LIN {X 0,Y 398.886,Z 784.107,A -85,B 0,C 180,E1 -11229.847,E2 -11229.847} C_VEL
LIN {X 0,Y 402.44,Z 816.531,A -85,B 0,C 180,E1 -11230.643,E2 -11230.643} C_VEL
LIN {X 0,Y 403.181,Z 824.962,A -85,B 0,C 180,E1 -11230.833,E2 -11230.833} C_VEL
LIN {X 0,Y 402.235,Z 895.243,A -85,B 0,C 180,E1 -11232.105,E2 -11232.105} C_VEL
LIN {X 0,Y 401.617,Z 908.446,A -85,B 0,C 180,E1 -11232.537,E2 -11232.537} C_VEL
LIN {X 0,Y 400.757,Z 921.743,A -85,B 0,C 180,E1 -11233.189,E2 -11233.189} C_VEL
LIN {X 0,Y 399.896,Z 932.958,A -85,B 0,C 180,E1 -11233.939,E2 -11233.939} C_VEL
LIN {X 0,Y 398.89,Z 944.652,A -85,B 0,C 180,E1 -11234.945,E2 -11234.945} C_VEL
LIN {X 0,Y 398.165,Z 954.79,A -85,B 0,C 180,E1 -11236.038,E2 -11236.038} C_VEL
LIN {X 0,Y 397.612,Z 963.944,A -85,B 0,C 180,E1 -11237.243,E2 -11237.243} C_VEL
LIN {X 0,Y 396.995,Z 971.973,A -85,B 0,C 180,E1 -11238.52,E2 -11238.52} C_VEL
LIN {X 0,Y 396.564,Z 979.861,A -85,B 0,C 180,E1 -11240.057,E2 -11240.057} C_VEL
LIN {X 0,Y 396.358,Z 987.17,A -85,B 0,C 180,E1 -11241.852,E2 -11241.852} C_VEL
LIN {X 0,Y 396.334,Z 991.594,A -85,B 0,C 180,E1 -11243.229,E2 -11243.229} C_VEL
LIN {X 0,Y 396.382,Z 995.807,A -85,B 0,C 180,E1 -11244.921,E2 -11244.921} C_VEL
LIN {X 0,Y 396.495,Z 997.753,A -85,B 0,C 180,E1 -11245.941,E2 -11245.941} C_VEL
LIN {X 0,Y 396.453,Z 999.193,A -85,B 0,C 180,E1 -11246.958,E2 -11246.958} C_VEL
LIN {X 0,Y 396.473,Z 1000.227,A -85,B 0,C 180,E1 -11247.975,E2 -11247.975} C_VEL
LIN {X 0,Y 396.505,Z 1000.858,A -85,B 0,C 180,E1 -11248.991,E2 -11248.991} C_VEL
LIN {X 0,Y 396.533,Z 1001.082,A -85,B 0,C 180,E1 -11250.007,E2 -11250.007} C_VEL
LIN {X 0,Y 396.505,Z 1000.85,A -85,B 0,C 180,E1 -11251.022,E2 -11251.022} C_VEL
LIN {X 0,Y 396.475,Z 1000.211,A -85,B 0,C 180,E1 -11252.038,E2 -11252.038} C_VEL
LIN {X 0,Y 396.455,Z 999.171,A -85,B 0,C 180,E1 -11253.055,E2 -11253.055} C_VEL
LIN {X 0,Y 396.499,Z 997.722,A -85,B 0,C 180,E1 -11254.072,E2 -11254.072} C_VEL
LIN {X 0,Y 396.305,Z 994.645,A -85,B 0,C 180,E1 -11255.604,E2 -11255.604} C_VEL
LIN {X 0,Y 396.296,Z 990.519,A -85,B 0,C 180,E1 -11257.137,E2 -11257.137} C_VEL
LIN {X 0,Y 396.416,Z 984.19,A -85,B 0,C 180,E1 -11258.93,E2 -11258.93} C_VEL
LIN {X 0,Y 396.65,Z 977.307,A -85,B 0,C 180,E1 -11260.47,E2 -11260.47} C_VEL
LIN {X 0,Y 397.201,Z 968.823,A -85,B 0,C 180,E1 -11262.005,E2 -11262.005} C_VEL
LIN {X 0,Y 397.865,Z 960.153,A -85,B 0,C 180,E1 -11263.282,E2 -11263.282} C_VEL
LIN {X 0,Y 398.568,Z 950.667,A -85,B 0,C 180,E1 -11264.428,E2 -11264.428} C_VEL
LIN {X 0,Y 399.272,Z 940.375,A -85,B 0,C 180,E1 -11265.446,E2 -11265.446} C_VEL
LIN {X 0,Y 400.17,Z 929.216,A -85,B 0,C 180,E1 -11266.326,E2 -11266.326} C_VEL
LIN {X 0,Y 401.098,Z 916.885,A -85,B 0,C 180,E1 -11267.073,E2 -11267.073} C_VEL
LIN {X 0,Y 401.822,Z 903.894,A -85,B 0,C 180,E1 -11267.632,E2 -11267.632} C_VEL
LIN {X 0,Y 402.351,Z 890.094,A -85,B 0,C 180,E1 -11268.002,E2 -11268.002} C_VEL
LIN {X 0,Y 403.048,Z 822.221,A -85,B 0,C 180,E1 -11269.218,E2 -11269.218} C_VEL
LIN {X 0,Y 400.233,Z 790.769,A -85,B 0,C 180,E1 -11270.212,E2 -11270.212} C_VEL
LIN {X 0,Y 399.008,Z 781.49,A -85,B 0,C 180,E1 -11270.565,E2 -11270.565} C_VEL
LIN {X 0,Y 400.608,Z 758.553,A -85,B 0,C 180,E1 -11274.181,E2 -11274.181} C_VEL
LIN {X 0,Y 402.329,Z 735.168,A -85,B 0,C 180,E1 -11277.863,E2 -11277.863} C_VEL
LIN {X 0,Y 402.724,Z 728.077,A -85,B 0,C 180,E1 -11278.999,E2 -11278.999} C_VEL
LIN {X 0,Y 399.691,Z 713.868,A -85,B 0,C 180,E1 -11281.546,E2 -11281.546} C_VEL
LIN {X 0,Y 397.055,Z 703.027,A -85,B 0,C 180,E1 -11283.615,E2 -11283.615} C_VEL
LIN {X 0,Y 397.093,Z 703.019,A -85,B 0,C 180,E1 -11287.208,E2 -11287.208} C_VEL
LIN {X 0,Y 397.072,Z 703.022,A -85,B 0,C 180,E1 -11290.44,E2 -11290.44} C_VEL
LIN {X 0,Y 397.058,Z 703.025,A -85,B 0,C 180,E1 -11293.66,E2 -11293.66} C_VEL
LIN {X 0,Y 397.108,Z 703.017,A -85,B 0,C 180,E1 -11296.526,E2 -11296.526} C_VEL
LIN {X 0,Y 397.104,Z 703.018,A -85,B 0,C 180,E1 -11300.422,E2 -11300.422} C_VEL
LIN {X 0,Y 397.111,Z 703.018,A -85,B 0,C 180,E1 -11303.006,E2 -11303.006} C_VEL
LIN {X 0,Y 397.13,Z 703.014,A -85,B 0,C 180,E1 -11306.728,E2 -11306.728} C_VEL
LIN {X 0,Y 397.135,Z 703.016,A -85,B 0,C 180,E1 -11310.297,E2 -11310.297} C_VEL
LIN {X 0,Y 397.104,Z 703.023,A -85,B 0,C 180,E1 -11313.739,E2 -11313.739} C_VEL
LIN {X 0,Y 397.121,Z 703.02,A -85,B 0,C 180,E1 -11317.086,E2 -11317.086} C_VEL
LIN {X 0,Y 397.139,Z 703.111,A -85,B 0,C 180,E1 -11319.435,E2 -11319.435} C_VEL
LIN {X 0,Y 398.123,Z 705.838,A -85,B 0,C 180,E1 -11319.602,E2 -11319.602} C_VEL
LIN {X 0,Y 402.78,Z 715.108,A -85,B 0,C 180,E1 -11320.252,E2 -11320.252} C_VEL
LIN {X 0,Y 405.375,Z 721.504,A -85,B 0,C 180,E1 -11320.626,E2 -11320.626} C_VEL
LIN {X 0,Y 403.629,Z 784.545,A -85,B 0,C 180,E1 -11322.161,E2 -11322.161} C_VEL
LIN {X 0,Y 403.565,Z 799.417,A -85,B 0,C 180,E1 -11322.681,E2 -11322.681} C_VEL
LIN {X 0,Y 403.241,Z 810.911,A -85,B 0,C 180,E1 -11323.268,E2 -11323.268} C_VEL
LIN {X 0,Y 402.848,Z 820.383,A -85,B 0,C 180,E1 -11323.886,E2 -11323.886} C_VEL
LIN {X 0,Y 402.399,Z 829.533,A -85,B 0,C 180,E1 -11324.622,E2 -11324.622} C_VEL
LIN {X 0,Y 401.801,Z 837.999,A -85,B 0,C 180,E1 -11325.437,E2 -11325.437} C_VEL
LIN {X 0,Y 401.36,Z 845.689,A -85,B 0,C 180,E1 -11326.326,E2 -11326.326} C_VEL
LIN {X 0,Y 400.76,Z 853.176,A -85,B 0,C 180,E1 -11327.337,E2 -11327.337} C_VEL
LIN {X 0,Y 400.089,Z 860.892,A -85,B 0,C 180,E1 -11328.602,E2 -11328.602} C_VEL
LIN {X 0,Y 399.508,Z 867.261,A -85,B 0,C 180,E1 -11329.868,E2 -11329.868} C_VEL
LIN {X 0,Y 399.059,Z 871.627,A -85,B 0,C 180,E1 -11330.88,E2 -11330.88} C_VEL
LIN {X 0,Y 398.612,Z 876.825,A -85,B 0,C 180,E1 -11332.401,E2 -11332.401} C_VEL
LIN {X 0,Y 397.936,Z 880.867,A -85,B 0,C 180,E1 -11333.917,E2 -11333.917} C_VEL
LIN {X 0,Y 397.839,Z 882.927,A -85,B 0,C 180,E1 -11334.933,E2 -11334.933} C_VEL
LIN {X 0,Y 397.507,Z 885.635,A -85,B 0,C 180,E1 -11336.96,E2 -11336.96} C_VEL
LIN {X 0,Y 397.313,Z 886.407,A -85,B 0,C 180,E1 -11337.973,E2 -11337.973} C_VEL
LIN {X 0,Y 397.23,Z 886.702,A -85,B 0,C 180,E1 -11338.986,E2 -11338.986} C_VEL
LIN {X 0,Y 397.162,Z 886.546,A -85,B 0,C 180,E1 -11340,E2 -11340} C_VEL
LIN {X 0,Y 397.162,Z 885.976,A -85,B 0,C 180,E1 -11341.014,E2 -11341.014} C_VEL
LIN {X 0,Y 396.969,Z 883.539,A -85,B 0,C 180,E1 -11343.045,E2 -11343.045} C_VEL
LIN {X 0,Y 397.213,Z 880.535,A -85,B 0,C 180,E1 -11344.567,E2 -11344.567} C_VEL
LIN {X 0,Y 397.481,Z 878.001,A -85,B 0,C 180,E1 -11345.581,E2 -11345.581} C_VEL
LIN {X 0,Y 397.666,Z 873.185,A -85,B 0,C 180,E1 -11347.106,E2 -11347.106} C_VEL
LIN {X 0,Y 398.012,Z 866.134,A -85,B 0,C 180,E1 -11348.821,E2 -11348.821} C_VEL
LIN {X 0,Y 398.382,Z 859.325,A -85,B 0,C 180,E1 -11350.161,E2 -11350.161} C_VEL
LIN {X 0,Y 398.726,Z 853.236,A -85,B 0,C 180,E1 -11351.18,E2 -11351.18} C_VEL
LIN {X 0,Y 399.083,Z 845.109,A -85,B 0,C 180,E1 -11352.329,E2 -11352.329} C_VEL
LIN {X 0,Y 399.579,Z 836.504,A -85,B 0,C 180,E1 -11353.347,E2 -11353.347} C_VEL
LIN {X 0,Y 399.983,Z 827.526,A -85,B 0,C 180,E1 -11354.24,E2 -11354.24} C_VEL
LIN {X 0,Y 400.347,Z 817.268,A -85,B 0,C 180,E1 -11355.081,E2 -11355.081} C_VEL
LIN {X 0,Y 400.669,Z 807.831,A -85,B 0,C 180,E1 -11355.711,E2 -11355.711} C_VEL
LIN {X 0,Y 400.901,Z 796.867,A -85,B 0,C 180,E1 -11356.289,E2 -11356.289} C_VEL
LIN {X 0,Y 401.134,Z 786.297,A -85,B 0,C 180,E1 -11356.705,E2 -11356.705} C_VEL
LIN {X 0,Y 401.245,Z 773.112,A -85,B 0,C 180,E1 -11357.061,E2 -11357.061} C_VEL
LIN {X 0,Y 402.038,Z 717.884,A -85,B 0,C 180,E1 -11358.241,E2 -11358.241} C_VEL
LIN {X 0,Y 397.183,Z 703.012,A -85,B 0,C 180,E1 -11358.773,E2 -11358.773} C_VEL
LIN {X 0,Y 397.113,Z 703.015,A -85,B 0,C 180,E1 -11361.818,E2 -11361.818} C_VEL
LIN {X 0,Y 397.12,Z 703.018,A -85,B 0,C 180,E1 -11365.134,E2 -11365.134} C_VEL
LIN {X 0,Y 397.092,Z 703.02,A -85,B 0,C 180,E1 -11368.546,E2 -11368.546} C_VEL
LIN {X 0,Y 397.099,Z 703.017,A -85,B 0,C 180,E1 -11371.834,E2 -11371.834} C_VEL
LIN {X 0,Y 397.136,Z 703.013,A -85,B 0,C 180,E1 -11374.493,E2 -11374.493} C_VEL
LIN {X 0,Y 397.11,Z 703.015,A -85,B 0,C 180,E1 -11378.274,E2 -11378.274} C_VEL
LIN {X 0,Y 397.07,Z 703.018,A -85,B 0,C 180,E1 -11381.974,E2 -11381.974} C_VEL
LIN {X 0,Y 397.104,Z 703.019,A -85,B 0,C 180,E1 -11385.067,E2 -11385.067} C_VEL
LIN {X 0,Y 397.069,Z 703.017,A -85,B 0,C 180,E1 -11388.021,E2 -11388.021} C_VEL
LIN {X 0,Y 397.107,Z 703.014,A -85,B 0,C 180,E1 -11391.72,E2 -11391.72} C_VEL
LIN {X 0,Y 397.132,Z 703.013,A -85,B 0,C 180,E1 -11395.502,E2 -11395.502} C_VEL
LIN {X 0,Y 397.088,Z 703.02,A -85,B 0,C 180,E1 -11399.113,E2 -11399.113} C_VEL
LIN {X 0,Y 397.072,Z 703.018,A -85,B 0,C 180,E1 -11402.249,E2 -11402.249} C_VEL
LIN {X 0,Y 397.115,Z 703.018,A -85,B 0,C 180,E1 -11404.86,E2 -11404.86} C_VEL
LIN {X 0,Y 397.1,Z 703.02,A -85,B 0,C 180,E1 -11408.176,E2 -11408.176} C_VEL
LIN {X 0,Y 397.155,Z 703.014,A -85,B 0,C 180,E1 -11410.303,E2 -11410.303} C_VEL
LIN {X 0,Y 398.938,Z 707.798,A -85,B 0,C 180,E1 -11410.502,E2 -11410.502} C_VEL
LIN {X 0,Y 404.02,Z 720.603,A -85,B 0,C 180,E1 -11411.009,E2 -11411.009} C_VEL
LIN {X 0,Y 403.44,Z 783.09,A -85,B 0,C 180,E1 -11412.147,E2 -11412.147} C_VEL
LIN {X 0,Y 403.437,Z 795.79,A -85,B 0,C 180,E1 -11412.539,E2 -11412.539} C_VEL
LIN {X 0,Y 403.11,Z 808.607,A -85,B 0,C 180,E1 -11413.146,E2 -11413.146} C_VEL
LIN {X 0,Y 402.546,Z 820.509,A -85,B 0,C 180,E1 -11413.913,E2 -11413.913} C_VEL
LIN {X 0,Y 401.957,Z 831.051,A -85,B 0,C 180,E1 -11414.79,E2 -11414.79} C_VEL
LIN {X 0,Y 401.223,Z 841.912,A -85,B 0,C 180,E1 -11415.928,E2 -11415.928} C_VEL
LIN {X 0,Y 400.613,Z 850.688,A -85,B 0,C 180,E1 -11417.069,E2 -11417.069} C_VEL
LIN {X 0,Y 399.894,Z 858.742,A -85,B 0,C 180,E1 -11418.334,E2 -11418.334} C_VEL
LIN {X 0,Y 399.146,Z 866.616,A -85,B 0,C 180,E1 -11419.853,E2 -11419.853} C_VEL
LIN {X 0,Y 398.615,Z 872.29,A -85,B 0,C 180,E1 -11421.209,E2 -11421.209} C_VEL
LIN {X 0,Y 398.205,Z 877.911,A -85,B 0,C 180,E1 -11422.897,E2 -11422.897} C_VEL
LIN {X 0,Y 397.689,Z 881.806,A -85,B 0,C 180,E1 -11424.416,E2 -11424.416} C_VEL
LIN {X 0,Y 397.543,Z 882.945,A -85,B 0,C 180,E1 -11424.976,E2 -11424.976} C_VEL
LIN {X 0,Y 396.731,Z 884.539,A -85,B 0,C 180,E1 -11425.794,E2 -11425.794} C_VEL
LIN {X 0,Y 393.77,Z 886.756,A -85,B 0,C 180,E1 -11427.128,E2 -11427.128} C_VEL
LIN {X 0,Y 391.337,Z 888.062,A -85,B 0,C 180,E1 -11428.216,E2 -11428.216} C_VEL
LIN {X 0,Y 390.213,Z 888.714,A -85,B 0,C 180,E1 -11429.211,E2 -11429.211} C_VEL
LIN {X 0,Y 390.184,Z 888.697,A -85,B 0,C 180,E1 -11429.355,E2 -11429.355} C_VEL
LIN {X 0,Y 390.223,Z 888.658,A -85,B 0,C 180,E1 -11431.025,E2 -11431.025} C_VEL
LIN {X 0,Y 390.329,Z 888.083,A -85,B 0,C 180,E1 -11432.057,E2 -11432.057} C_VEL
LIN {X 0,Y 390.339,Z 885.852,A -85,B 0,C 180,E1 -11434.123,E2 -11434.123} C_VEL
LIN {X 0,Y 390.687,Z 883.043,A -85,B 0,C 180,E1 -11435.671,E2 -11435.671} C_VEL
LIN {X 0,Y 391.201,Z 879.222,A -85,B 0,C 180,E1 -11437.217,E2 -11437.217} C_VEL
LIN {X 0,Y 391.648,Z 873.751,A -85,B 0,C 180,E1 -11438.928,E2 -11438.928} C_VEL
LIN {X 0,Y 392.316,Z 866.944,A -85,B 0,C 180,E1 -11440.573,E2 -11440.573} C_VEL
LIN {X 0,Y 393.147,Z 858.923,A -85,B 0,C 180,E1 -11442.117,E2 -11442.117} C_VEL
LIN {X 0,Y 393.866,Z 850.708,A -85,B 0,C 180,E1 -11443.405,E2 -11443.405} C_VEL
LIN {X 0,Y 394.611,Z 840.549,A -85,B 0,C 180,E1 -11444.694,E2 -11444.694} C_VEL
LIN {X 0,Y 395.431,Z 830.092,A -85,B 0,C 180,E1 -11445.752,E2 -11445.752} C_VEL
LIN {X 0,Y 396.049,Z 818.837,A -85,B 0,C 180,E1 -11446.662,E2 -11446.662} C_VEL
LIN {X 0,Y 396.497,Z 806.955,A -85,B 0,C 180,E1 -11447.396,E2 -11447.396} C_VEL
LIN {X 0,Y 396.707,Z 793.593,A -85,B 0,C 180,E1 -11447.986,E2 -11447.986} C_VEL
LIN {X 0,Y 396.795,Z 780.202,A -85,B 0,C 180,E1 -11448.349,E2 -11448.349} C_VEL
LIN {X 0,Y 397.353,Z 722.142,A -85,B 0,C 180,E1 -11449.413,E2 -11449.413} C_VEL
LIN {X 0,Y 390.141,Z 704.2,A -85,B 0,C 180,E1 -11450.154,E2 -11450.154} C_VEL
LIN {X 0,Y 390.093,Z 703.895,A -85,B 0,C 180,E1 -11450.215,E2 -11450.215} C_VEL
LIN {X 0,Y 390.068,Z 703.894,A -85,B 0,C 180,E1 -11453.343,E2 -11453.343} C_VEL
LIN {X 0,Y 390.088,Z 703.889,A -85,B 0,C 180,E1 -11456.76,E2 -11456.76} C_VEL
LIN {X 0,Y 390.01,Z 703.899,A -85,B 0,C 180,E1 -11460.292,E2 -11460.292} C_VEL
LIN {X 0,Y 390.035,Z 703.896,A -85,B 0,C 180,E1 -11464.017,E2 -11464.017} C_VEL
LIN {X 0,Y 390.01,Z 703.893,A -85,B 0,C 180,E1 -11467.544,E2 -11467.544} C_VEL
LIN {X 0,Y 390.042,Z 703.899,A -85,B 0,C 180,E1 -11470.818,E2 -11470.818} C_VEL
LIN {X 0,Y 390.085,Z 703.883,A -85,B 0,C 180,E1 -11473.89,E2 -11473.89} C_VEL
LIN {X 0,Y 390.07,Z 703.888,A -85,B 0,C 180,E1 -11476.791,E2 -11476.791} C_VEL
LIN {X 0,Y 390.028,Z 703.905,A -85,B 0,C 180,E1 -11479.557,E2 -11479.557} C_VEL
LIN {X 0,Y 389.994,Z 703.904,A -85,B 0,C 180,E1 -11482.442,E2 -11482.442} C_VEL
LIN {X 0,Y 390.011,Z 703.899,A -85,B 0,C 180,E1 -11486.039,E2 -11486.039} C_VEL
LIN {X 0,Y 389.988,Z 703.904,A -85,B 0,C 180,E1 -11488.492,E2 -11488.492} C_VEL
LIN {X 0,Y 390.056,Z 703.893,A -85,B 0,C 180,E1 -11492.065,E2 -11492.065} C_VEL
LIN {X 0,Y 390.015,Z 703.897,A -85,B 0,C 180,E1 -11495.515,E2 -11495.515} C_VEL
LIN {X 0,Y 389.995,Z 703.904,A -85,B 0,C 180,E1 -11498.874,E2 -11498.874} C_VEL
LIN {X 0,Y 390.059,Z 703.891,A -85,B 0,C 180,E1 -11502.163,E2 -11502.163} C_VEL
LIN {X 0,Y 390.08,Z 703.892,A -85,B 0,C 180,E1 -11505.39,E2 -11505.39} C_VEL
LIN {X 0,Y 390.09,Z 703.888,A -85,B 0,C 180,E1 -11508.569,E2 -11508.569} C_VEL
LIN {X 0,Y 390.236,Z 703.874,A -85,B 0,C 180,E1 -11512.03,E2 -11512.03} C_VEL
LIN {X 0,Y 390.163,Z 703.882,A -85,B 0,C 180,E1 -11514.833,E2 -11514.833} C_VEL
LIN {X 0,Y 390.349,Z 703.859,A -85,B 0,C 180,E1 -11517.936,E2 -11517.936} C_VEL
LIN {X 0,Y 390.478,Z 703.845,A -85,B 0,C 180,E1 -11520,E2 -11520} C_VEL
LIN {X 0,Y 390.278,Z 703.865,A -85,B 0,C 180,E1 -11523.097,E2 -11523.097} C_VEL
LIN {X 0,Y 390.265,Z 703.871,A -85,B 0,C 180,E1 -11526.203,E2 -11526.203} C_VEL
LIN {X 0,Y 390.139,Z 703.882,A -85,B 0,C 180,E1 -11529.33,E2 -11529.33} C_VEL
LIN {X 0,Y 390.108,Z 703.889,A -85,B 0,C 180,E1 -11532.485,E2 -11532.485} C_VEL
LIN {X 0,Y 390.075,Z 703.896,A -85,B 0,C 180,E1 -11535.68,E2 -11535.68} C_VEL
LIN {X 0,Y 390.036,Z 703.898,A -85,B 0,C 180,E1 -11538.926,E2 -11538.926} C_VEL
LIN {X 0,Y 389.973,Z 703.905,A -85,B 0,C 180,E1 -11542.238,E2 -11542.238} C_VEL
LIN {X 0,Y 390.056,Z 703.892,A -85,B 0,C 180,E1 -11545.748,E2 -11545.748} C_VEL
LIN {X 0,Y 390.003,Z 703.901,A -85,B 0,C 180,E1 -11549.114,E2 -11549.114} C_VEL
LIN {X 0,Y 389.997,Z 703.902,A -85,B 0,C 180,E1 -11552.726,E2 -11552.726} C_VEL
LIN {X 0,Y 390.002,Z 703.905,A -85,B 0,C 180,E1 -11555.831,E2 -11555.831} C_VEL
LIN {X 0,Y 390.023,Z 703.888,A -85,B 0,C 180,E1 -11559.226,E2 -11559.226} C_VEL
LIN {X 0,Y 390.072,Z 703.896,A -85,B 0,C 180,E1 -11562.393,E2 -11562.393} C_VEL
LIN {X 0,Y 390.073,Z 703.893,A -85,B 0,C 180,E1 -11565.372,E2 -11565.372} C_VEL
LIN {X 0,Y 390.063,Z 703.891,A -85,B 0,C 180,E1 -11568.204,E2 -11568.204} C_VEL
LIN {X 0,Y 390.055,Z 703.894,A -85,B 0,C 180,E1 -11570.916,E2 -11570.916} C_VEL
LIN {X 0,Y 390.05,Z 703.898,A -85,B 0,C 180,E1 -11574.801,E2 -11574.801} C_VEL
LIN {X 0,Y 390.068,Z 703.973,A -85,B 0,C 180,E1 -11576.056,E2 -11576.056} C_VEL
LIN {X 0,Y 394.349,Z 722.022,A -85,B 0,C 180,E1 -11579.489,E2 -11579.489} C_VEL
LIN {X 0,Y 395.934,Z 729.889,A -85,B 0,C 180,E1 -11580.908,E2 -11580.908} C_VEL
LIN {X 0,Y 394.456,Z 748.1,A -85,B 0,C 180,E1 -11583.844,E2 -11583.844} C_VEL
LIN {X 0,Y 392.968,Z 768.475,A -85,B 0,C 180,E1 -11587.118,E2 -11587.118} C_VEL
LIN {X 0,Y 391.958,Z 783.231,A -85,B 0,C 180,E1 -11589.5,E2 -11589.5} C_VEL
LIN {X 0,Y 395.427,Z 814.793,A -85,B 0,C 180,E1 -11590.272,E2 -11590.272} C_VEL
LIN {X 0,Y 396.462,Z 826.067,A -85,B 0,C 180,E1 -11590.534,E2 -11590.534} C_VEL
LIN {X 0,Y 395.468,Z 894.24,A -85,B 0,C 180,E1 -11591.789,E2 -11591.789} C_VEL
LIN {X 0,Y 394.839,Z 907.44,A -85,B 0,C 180,E1 -11592.228,E2 -11592.228} C_VEL
LIN {X 0,Y 393.921,Z 920.729,A -85,B 0,C 180,E1 -11592.888,E2 -11592.888} C_VEL
LIN {X 0,Y 393.035,Z 931.942,A -85,B 0,C 180,E1 -11593.651,E2 -11593.651} C_VEL
LIN {X 0,Y 392.038,Z 943.642,A -85,B 0,C 180,E1 -11594.676,E2 -11594.676} C_VEL
LIN {X 0,Y 391.184,Z 954.338,A -85,B 0,C 180,E1 -11595.853,E2 -11595.853} C_VEL
LIN {X 0,Y 390.668,Z 962.93,A -85,B 0,C 180,E1 -11597.013,E2 -11597.013} C_VEL
LIN {X 0,Y 389.977,Z 970.953,A -85,B 0,C 180,E1 -11598.31,E2 -11598.31} C_VEL
LIN {X 0,Y 389.51,Z 978.841,A -85,B 0,C 180,E1 -11599.875,E2 -11599.875} C_VEL
LIN {X 0,Y 389.279,Z 986.151,A -85,B 0,C 180,E1 -11601.703,E2 -11601.703} C_VEL
LIN {X 0,Y 389.275,Z 990.867,A -85,B 0,C 180,E1 -11603.206,E2 -11603.206} C_VEL
LIN {X 0,Y 389.302,Z 994.793,A -85,B 0,C 180,E1 -11604.828,E2 -11604.828} C_VEL
LIN {X 0,Y 389.44,Z 996.744,A -85,B 0,C 180,E1 -11605.868,E2 -11605.868} C_VEL
LIN {X 0,Y 389.411,Z 998.187,A -85,B 0,C 180,E1 -11606.903,E2 -11606.903} C_VEL
LIN {X 0,Y 389.434,Z 999.222,A -85,B 0,C 180,E1 -11607.939,E2 -11607.939} C_VEL
LIN {X 0,Y 389.471,Z 999.855,A -85,B 0,C 180,E1 -11608.973,E2 -11608.973} C_VEL
LIN {X 0,Y 389.504,Z 1000.079,A -85,B 0,C 180,E1 -11610.007,E2 -11610.007} C_VEL
LIN {X 0,Y 389.472,Z 999.846,A -85,B 0,C 180,E1 -11611.041,E2 -11611.041} C_VEL
LIN {X 0,Y 389.435,Z 999.206,A -85,B 0,C 180,E1 -11612.075,E2 -11612.075} C_VEL
LIN {X 0,Y 389.414,Z 998.164,A -85,B 0,C 180,E1 -11613.11,E2 -11613.11} C_VEL
LIN {X 0,Y 389.444,Z 996.712,A -85,B 0,C 180,E1 -11614.146,E2 -11614.146} C_VEL
LIN {X 0,Y 389.243,Z 993.632,A -85,B 0,C 180,E1 -11615.706,E2 -11615.706} C_VEL
LIN {X 0,Y 389.233,Z 989.502,A -85,B 0,C 180,E1 -11617.268,E2 -11617.268} C_VEL
LIN {X 0,Y 389.35,Z 983.168,A -85,B 0,C 180,E1 -11619.094,E2 -11619.094} C_VEL
LIN {X 0,Y 389.626,Z 976.286,A -85,B 0,C 180,E1 -11620.661,E2 -11620.661} C_VEL
LIN {X 0,Y 390.154,Z 967.793,A -85,B 0,C 180,E1 -11622.226,E2 -11622.226} C_VEL
LIN {X 0,Y 390.802,Z 959.115,A -85,B 0,C 180,E1 -11623.526,E2 -11623.526} C_VEL
LIN {X 0,Y 391.733,Z 948.45,A -85,B 0,C 180,E1 -11624.818,E2 -11624.818} C_VEL
LIN {X 0,Y 392.419,Z 939.356,A -85,B 0,C 180,E1 -11625.723,E2 -11625.723} C_VEL
LIN {X 0,Y 393.314,Z 928.191,A -85,B 0,C 180,E1 -11626.618,E2 -11626.618} C_VEL
LIN {X 0,Y 394.306,Z 915.864,A -85,B 0,C 180,E1 -11627.376,E2 -11627.376} C_VEL
LIN {X 0,Y 395.059,Z 902.871,A -85,B 0,C 180,E1 -11627.944,E2 -11627.944} C_VEL
LIN {X 0,Y 395.553,Z 889.057,A -85,B 0,C 180,E1 -11628.322,E2 -11628.322} C_VEL
LIN {X 0,Y 396.433,Z 829.277,A -85,B 0,C 180,E1 -11629.43,E2 -11629.43} C_VEL
LIN {X 0,Y 396.382,Z 821.582,A -85,B 0,C 180,E1 -11629.638,E2 -11629.638} C_VEL
LIN {X 0,Y 393.881,Z 791.903,A -85,B 0,C 180,E1 -11630.636,E2 -11630.636} C_VEL
LIN {X 0,Y 392.211,Z 779.278,A -85,B 0,C 180,E1 -11631.134,E2 -11631.134} C_VEL
LIN {X 0,Y 393.727,Z 758.008,A -85,B 0,C 180,E1 -11634.557,E2 -11634.557} C_VEL
LIN {X 0,Y 395.46,Z 735.94,A -85,B 0,C 180,E1 -11638.102,E2 -11638.102} C_VEL
LIN {X 0,Y 395.85,Z 729.808,A -85,B 0,C 180,E1 -11639.1,E2 -11639.1} C_VEL
LIN {X 0,Y 393.035,Z 716.425,A -85,B 0,C 180,E1 -11641.541,E2 -11641.541} C_VEL
LIN {X 0,Y 390.014,Z 703.908,A -85,B 0,C 180,E1 -11643.966,E2 -11643.966} C_VEL
LIN {X 0,Y 390.047,Z 703.899,A -85,B 0,C 180,E1 -11647.785,E2 -11647.785} C_VEL
LIN {X 0,Y 390.033,Z 703.899,A -85,B 0,C 180,E1 -11650.817,E2 -11650.817} C_VEL
LIN {X 0,Y 390.007,Z 703.902,A -85,B 0,C 180,E1 -11653.879,E2 -11653.879} C_VEL
LIN {X 0,Y 390.064,Z 703.895,A -85,B 0,C 180,E1 -11656.79,E2 -11656.79} C_VEL
LIN {X 0,Y 390.028,Z 703.903,A -85,B 0,C 180,E1 -11659.557,E2 -11659.557} C_VEL
LIN {X 0,Y 390.056,Z 703.896,A -85,B 0,C 180,E1 -11662.453,E2 -11662.453} C_VEL
LIN {X 0,Y 390.081,Z 703.893,A -85,B 0,C 180,E1 -11666.046,E2 -11666.046} C_VEL
LIN {X 0,Y 390.062,Z 703.896,A -85,B 0,C 180,E1 -11669.872,E2 -11669.872} C_VEL
LIN {X 0,Y 390.064,Z 703.898,A -85,B 0,C 180,E1 -11673.228,E2 -11673.228} C_VEL
LIN {X 0,Y 390.086,Z 703.895,A -85,B 0,C 180,E1 -11676.766,E2 -11676.766} C_VEL
LIN {X 0,Y 390.07,Z 703.897,A -85,B 0,C 180,E1 -11678.827,E2 -11678.827} C_VEL
LIN {X 0,Y 391.247,Z 707.02,A -85,B 0,C 180,E1 -11679.039,E2 -11679.039} C_VEL
LIN {X 0,Y 396.787,Z 717.894,A -85,B 0,C 180,E1 -11679.851,E2 -11679.851} C_VEL
LIN {X 0,Y 398.929,Z 722.919,A -85,B 0,C 180,E1 -11680.178,E2 -11680.178} C_VEL
LIN {X 0,Y 397.675,Z 763.334,A -85,B 0,C 180,E1 -11681.2,E2 -11681.2} C_VEL
LIN {X 0,Y 397.159,Z 789.992,A -85,B 0,C 180,E1 -11681.894,E2 -11681.894} C_VEL
LIN {X 0,Y 397.028,Z 802.372,A -85,B 0,C 180,E1 -11682.387,E2 -11682.387} C_VEL
LIN {X 0,Y 396.71,Z 812.257,A -85,B 0,C 180,E1 -11682.911,E2 -11682.911} C_VEL
LIN {X 0,Y 396.271,Z 822.276,A -85,B 0,C 180,E1 -11683.582,E2 -11683.582} C_VEL
LIN {X 0,Y 395.787,Z 831.378,A -85,B 0,C 180,E1 -11684.336,E2 -11684.336} C_VEL
LIN {X 0,Y 395.169,Z 839.944,A -85,B 0,C 180,E1 -11685.187,E2 -11685.187} C_VEL
LIN {X 0,Y 394.693,Z 847.522,A -85,B 0,C 180,E1 -11686.091,E2 -11686.091} C_VEL
LIN {X 0,Y 394.034,Z 854.879,A -85,B 0,C 180,E1 -11687.118,E2 -11687.118} C_VEL
LIN {X 0,Y 393.316,Z 862.474,A -85,B 0,C 180,E1 -11688.403,E2 -11688.403} C_VEL
LIN {X 0,Y 392.701,Z 868.76,A -85,B 0,C 180,E1 -11689.69,E2 -11689.69} C_VEL
LIN {X 0,Y 392.201,Z 873.088,A -85,B 0,C 180,E1 -11690.719,E2 -11690.719} C_VEL
LIN {X 0,Y 391.711,Z 878.224,A -85,B 0,C 180,E1 -11692.267,E2 -11692.267} C_VEL
LIN {X 0,Y 391.017,Z 882.206,A -85,B 0,C 180,E1 -11693.809,E2 -11693.809} C_VEL
LIN {X 0,Y 390.902,Z 884.255,A -85,B 0,C 180,E1 -11694.842,E2 -11694.842} C_VEL
LIN {X 0,Y 390.52,Z 886.834,A -85,B 0,C 180,E1 -11696.905,E2 -11696.905} C_VEL
LIN {X 0,Y 390.339,Z 887.58,A -85,B 0,C 180,E1 -11697.936,E2 -11697.936} C_VEL
LIN {X 0,Y 390.219,Z 887.812,A -85,B 0,C 180,E1 -11698.968,E2 -11698.968} C_VEL
LIN {X 0,Y 390.144,Z 887.614,A -85,B 0,C 180,E1 -11700,E2 -11700} C_VEL
LIN {X 0,Y 390.141,Z 887.009,A -85,B 0,C 180,E1 -11701.032,E2 -11701.032} C_VEL
LIN {X 0,Y 389.939,Z 884.457,A -85,B 0,C 180,E1 -11703.1,E2 -11703.1} C_VEL
LIN {X 0,Y 390.201,Z 881.368,A -85,B 0,C 180,E1 -11704.649,E2 -11704.649} C_VEL
LIN {X 0,Y 390.451,Z 878.787,A -85,B 0,C 180,E1 -11705.682,E2 -11705.682} C_VEL
LIN {X 0,Y 390.742,Z 872.839,A -85,B 0,C 180,E1 -11707.493,E2 -11707.493} C_VEL
LIN {X 0,Y 391.018,Z 866.344,A -85,B 0,C 180,E1 -11709.048,E2 -11709.048} C_VEL
LIN {X 0,Y 391.405,Z 859.725,A -85,B 0,C 180,E1 -11710.344,E2 -11710.344} C_VEL
LIN {X 0,Y 391.757,Z 853.492,A -85,B 0,C 180,E1 -11711.381,E2 -11711.381} C_VEL
LIN {X 0,Y 392.158,Z 845.2,A -85,B 0,C 180,E1 -11712.55,E2 -11712.55} C_VEL
LIN {X 0,Y 392.567,Z 837.62,A -85,B 0,C 180,E1 -11713.458,E2 -11713.458} C_VEL
LIN {X 0,Y 392.999,Z 828.647,A -85,B 0,C 180,E1 -11714.367,E2 -11714.367} C_VEL
LIN {X 0,Y 393.352,Z 819.753,A -85,B 0,C 180,E1 -11715.123,E2 -11715.123} C_VEL
LIN {X 0,Y 393.698,Z 808.997,A -85,B 0,C 180,E1 -11715.864,E2 -11715.864} C_VEL
LIN {X 0,Y 393.927,Z 798.09,A -85,B 0,C 180,E1 -11716.453,E2 -11716.453} C_VEL
LIN {X 0,Y 394.166,Z 787.645,A -85,B 0,C 180,E1 -11716.876,E2 -11716.876} C_VEL
LIN {X 0,Y 394.332,Z 774.744,A -85,B 0,C 180,E1 -11717.236,E2 -11717.236} C_VEL
LIN {X 0,Y 395.125,Z 719.239,A -85,B 0,C 180,E1 -11718.459,E2 -11718.459} C_VEL
LIN {X 0,Y 390.127,Z 703.891,A -85,B 0,C 180,E1 -11719.024,E2 -11719.024} C_VEL
LIN {X 0,Y 390.054,Z 703.895,A -85,B 0,C 180,E1 -11722.233,E2 -11722.233} C_VEL
LIN {X 0,Y 390.07,Z 703.893,A -85,B 0,C 180,E1 -11725.721,E2 -11725.721} C_VEL
LIN {X 0,Y 390.049,Z 703.899,A -85,B 0,C 180,E1 -11729.11,E2 -11729.11} C_VEL
LIN {X 0,Y 390.06,Z 703.899,A -85,B 0,C 180,E1 -11732.72,E2 -11732.72} C_VEL
LIN {X 0,Y 390.062,Z 703.892,A -85,B 0,C 180,E1 -11735.82,E2 -11735.82} C_VEL
LIN {X 0,Y 390.056,Z 703.897,A -85,B 0,C 180,E1 -11739.21,E2 -11739.21} C_VEL
LIN {X 0,Y 390.049,Z 703.893,A -85,B 0,C 180,E1 -11742.369,E2 -11742.369} C_VEL
LIN {X 0,Y 390.06,Z 703.894,A -85,B 0,C 180,E1 -11745.351,E2 -11745.351} C_VEL
LIN {X 0,Y 390.033,Z 703.894,A -85,B 0,C 180,E1 -11748.181,E2 -11748.181} C_VEL
LIN {X 0,Y 390.075,Z 703.893,A -85,B 0,C 180,E1 -11750.9,E2 -11750.9} C_VEL
LIN {X 0,Y 390.085,Z 703.891,A -85,B 0,C 180,E1 -11754.788,E2 -11754.788} C_VEL
LIN {X 0,Y 390.033,Z 703.895,A -85,B 0,C 180,E1 -11758.491,E2 -11758.491} C_VEL
LIN {X 0,Y 390.032,Z 703.896,A -85,B 0,C 180,E1 -11761.999,E2 -11761.999} C_VEL
LIN {X 0,Y 390.05,Z 703.899,A -85,B 0,C 180,E1 -11765.512,E2 -11765.512} C_VEL
LIN {X 0,Y 390.061,Z 703.899,A -85,B 0,C 180,E1 -11768.872,E2 -11768.872} C_VEL
LIN {X 0,Y 390.11,Z 703.893,A -85,B 0,C 180,E1 -11769.938,E2 -11769.938} C_VEL
LIN {X 0,Y 391.72,Z 708.323,A -85,B 0,C 180,E1 -11770.116,E2 -11770.116} C_VEL
LIN {X 0,Y 397.403,Z 722.438,A -85,B 0,C 180,E1 -11770.696,E2 -11770.696} C_VEL
LIN {X 0,Y 396.736,Z 784.117,A -85,B 0,C 180,E1 -11771.835,E2 -11771.835} C_VEL
LIN {X 0,Y 396.728,Z 796.807,A -85,B 0,C 180,E1 -11772.234,E2 -11772.234} C_VEL
LIN {X 0,Y 396.385,Z 809.619,A -85,B 0,C 180,E1 -11772.851,E2 -11772.851} C_VEL
LIN {X 0,Y 395.798,Z 821.516,A -85,B 0,C 180,E1 -11773.631,E2 -11773.631} C_VEL
LIN {X 0,Y 395.18,Z 832.058,A -85,B 0,C 180,E1 -11774.522,E2 -11774.522} C_VEL
LIN {X 0,Y 394.41,Z 842.919,A -85,B 0,C 180,E1 -11775.68,E2 -11775.68} C_VEL
LIN {X 0,Y 393.766,Z 851.694,A -85,B 0,C 180,E1 -11776.84,E2 -11776.84} C_VEL
LIN {X 0,Y 393.018,Z 859.747,A -85,B 0,C 180,E1 -11778.127,E2 -11778.127} C_VEL
LIN {X 0,Y 392.23,Z 867.621,A -85,B 0,C 180,E1 -11779.672,E2 -11779.672} C_VEL
LIN {X 0,Y 391.671,Z 873.293,A -85,B 0,C 180,E1 -11781.051,E2 -11781.051} C_VEL
LIN {X 0,Y 391.236,Z 878.914,A -85,B 0,C 180,E1 -11782.77,E2 -11782.77} C_VEL
LIN {X 0,Y 390.697,Z 882.81,A -85,B 0,C 180,E1 -11784.316,E2 -11784.316} C_VEL
LIN {X 0,Y 390.352,Z 885.676,A -85,B 0,C 180,E1 -11785.864,E2 -11785.864} C_VEL
LIN {X 0,Y 390.311,Z 887.037,A -85,B 0,C 180,E1 -11786.897,E2 -11786.897} C_VEL
LIN {X 0,Y 390.309,Z 888,A -85,B 0,C 180,E1 -11787.929,E2 -11787.929} C_VEL
LIN {X 0,Y 390.184,Z 888.697,A -85,B 0,C 180,E1 -11789.355,E2 -11789.355} C_VEL
LIN {X 0,Y 389.497,Z 888.922,A -85,B 0,C 180,E1 -11790.218,E2 -11790.218} C_VEL
LIN {X 0,Y 386.677,Z 888.906,A -85,B 0,C 180,E1 -11791.622,E2 -11791.622} C_VEL
LIN {X 0,Y 384.336,Z 888.405,A -85,B 0,C 180,E1 -11792.752,E2 -11792.752} C_VEL
LIN {X 0,Y 383.366,Z 887.61,A -85,B 0,C 180,E1 -11793.619,E2 -11793.619} C_VEL
LIN {X 0,Y 383.305,Z 887.212,A -85,B 0,C 180,E1 -11793.911,E2 -11793.911} C_VEL
LIN {X 0,Y 383.695,Z 884.044,A -85,B 0,C 180,E1 -11795.774,E2 -11795.774} C_VEL
LIN {X 0,Y 384.234,Z 880.223,A -85,B 0,C 180,E1 -11797.349,E2 -11797.349} C_VEL
LIN {X 0,Y 384.707,Z 874.752,A -85,B 0,C 180,E1 -11799.09,E2 -11799.09} C_VEL
LIN {X 0,Y 385.409,Z 867.944,A -85,B 0,C 180,E1 -11800.765,E2 -11800.765} C_VEL
LIN {X 0,Y 386.28,Z 859.922,A -85,B 0,C 180,E1 -11802.336,E2 -11802.336} C_VEL
LIN {X 0,Y 387.033,Z 851.707,A -85,B 0,C 180,E1 -11803.646,E2 -11803.646} C_VEL
LIN {X 0,Y 387.817,Z 841.548,A -85,B 0,C 180,E1 -11804.957,E2 -11804.957} C_VEL
LIN {X 0,Y 388.68,Z 831.088,A -85,B 0,C 180,E1 -11806.033,E2 -11806.033} C_VEL
LIN {X 0,Y 389.321,Z 819.833,A -85,B 0,C 180,E1 -11806.958,E2 -11806.958} C_VEL
LIN {X 0,Y 389.788,Z 807.95,A -85,B 0,C 180,E1 -11807.705,E2 -11807.705} C_VEL
LIN {X 0,Y 390.035,Z 795.486,A -85,B 0,C 180,E1 -11808.27,E2 -11808.27} C_VEL
LIN {X 0,Y 390.13,Z 782.749,A -85,B 0,C 180,E1 -11808.64,E2 -11808.64} C_VEL
LIN {X 0,Y 390.66,Z 733.984,A -85,B 0,C 180,E1 -11809.551,E2 -11809.551} C_VEL
LIN {X 0,Y 390.566,Z 723.47,A -85,B 0,C 180,E1 -11809.758,E2 -11809.758} C_VEL
LIN {X 0,Y 383.083,Z 705.135,A -85,B 0,C 180,E1 -11810.544,E2 -11810.544} C_VEL
LIN {X 0,Y 383.04,Z 704.773,A -85,B 0,C 180,E1 -11810.604,E2 -11810.604} C_VEL
LIN {X 0,Y 383.011,Z 704.771,A -85,B 0,C 180,E1 -11813.799,E2 -11813.799} C_VEL
LIN {X 0,Y 383.055,Z 704.762,A -85,B 0,C 180,E1 -11816.115,E2 -11816.115} C_VEL
LIN {X 0,Y 382.964,Z 704.778,A -85,B 0,C 180,E1 -11819.692,E2 -11819.692} C_VEL
LIN {X 0,Y 382.971,Z 704.782,A -85,B 0,C 180,E1 -11823.393,E2 -11823.393} C_VEL
LIN {X 0,Y 382.998,Z 704.775,A -85,B 0,C 180,E1 -11826.157,E2 -11826.157} C_VEL
LIN {X 0,Y 382.981,Z 704.78,A -85,B 0,C 180,E1 -11829.949,E2 -11829.949} C_VEL
LIN {X 0,Y 383.023,Z 704.773,A -85,B 0,C 180,E1 -11832.781,E2 -11832.781} C_VEL
LIN {X 0,Y 383.026,Z 704.759,A -85,B 0,C 180,E1 -11835.793,E2 -11835.793} C_VEL
LIN {X 0,Y 382.995,Z 704.776,A -85,B 0,C 180,E1 -11838.78,E2 -11838.78} C_VEL
LIN {X 0,Y 382.951,Z 704.783,A -85,B 0,C 180,E1 -11842.089,E2 -11842.089} C_VEL
LIN {X 0,Y 382.962,Z 704.777,A -85,B 0,C 180,E1 -11845.326,E2 -11845.326} C_VEL
LIN {X 0,Y 382.978,Z 704.779,A -85,B 0,C 180,E1 -11847.847,E2 -11847.847} C_VEL
LIN {X 0,Y 382.992,Z 704.769,A -85,B 0,C 180,E1 -11851.718,E2 -11851.718} C_VEL
LIN {X 0,Y 382.988,Z 704.772,A -85,B 0,C 180,E1 -11855.035,E2 -11855.035} C_VEL
LIN {X 0,Y 382.932,Z 704.787,A -85,B 0,C 180,E1 -11858.465,E2 -11858.465} C_VEL
LIN {X 0,Y 382.994,Z 704.771,A -85,B 0,C 180,E1 -11861.823,E2 -11861.823} C_VEL
LIN {X 0,Y 383.046,Z 704.77,A -85,B 0,C 180,E1 -11865.116,E2 -11865.116} C_VEL
LIN {X 0,Y 383.039,Z 704.769,A -85,B 0,C 180,E1 -11868.356,E2 -11868.356} C_VEL
LIN {X 0,Y 383.193,Z 704.751,A -85,B 0,C 180,E1 -11871.973,E2 -11871.973} C_VEL
LIN {X 0,Y 383.135,Z 704.759,A -85,B 0,C 180,E1 -11874.738,E2 -11874.738} C_VEL
LIN {X 0,Y 383.318,Z 704.735,A -85,B 0,C 180,E1 -11877.898,E2 -11877.898} C_VEL
LIN {X 0,Y 383.448,Z 704.721,A -85,B 0,C 180,E1 -11880,E2 -11880} C_VEL
LIN {X 0,Y 383.213,Z 704.745,A -85,B 0,C 180,E1 -11883.154,E2 -11883.154} C_VEL
LIN {X 0,Y 383.219,Z 704.749,A -85,B 0,C 180,E1 -11886.317,E2 -11886.317} C_VEL
LIN {X 0,Y 383.086,Z 704.761,A -85,B 0,C 180,E1 -11889.504,E2 -11889.504} C_VEL
LIN {X 0,Y 383.072,Z 704.767,A -85,B 0,C 180,E1 -11892.718,E2 -11892.718} C_VEL
LIN {X 0,Y 383.015,Z 704.772,A -85,B 0,C 180,E1 -11895.976,E2 -11895.976} C_VEL
LIN {X 0,Y 382.991,Z 704.779,A -85,B 0,C 180,E1 -11899.287,E2 -11899.287} C_VEL
LIN {X 0,Y 382.942,Z 704.779,A -85,B 0,C 180,E1 -11902.669,E2 -11902.669} C_VEL
LIN {X 0,Y 383.017,Z 704.769,A -85,B 0,C 180,E1 -11906.128,E2 -11906.128} C_VEL
LIN {X 0,Y 382.988,Z 704.775,A -85,B 0,C 180,E1 -11908.497,E2 -11908.497} C_VEL
LIN {X 0,Y 382.95,Z 704.781,A -85,B 0,C 180,E1 -11912.433,E2 -11912.433} C_VEL
LIN {X 0,Y 382.971,Z 704.783,A -85,B 0,C 180,E1 -11915.962,E2 -11915.962} C_VEL
LIN {X 0,Y 382.971,Z 704.767,A -85,B 0,C 180,E1 -11919.594,E2 -11919.594} C_VEL
LIN {X 0,Y 383.018,Z 704.774,A -85,B 0,C 180,E1 -11922.795,E2 -11922.795} C_VEL
LIN {X 0,Y 383.027,Z 704.773,A -85,B 0,C 180,E1 -11925.807,E2 -11925.807} C_VEL
LIN {X 0,Y 383.003,Z 704.778,A -85,B 0,C 180,E1 -11928.794,E2 -11928.794} C_VEL
LIN {X 0,Y 382.965,Z 704.783,A -85,B 0,C 180,E1 -11932.103,E2 -11932.103} C_VEL
LIN {X 0,Y 382.991,Z 704.766,A -85,B 0,C 180,E1 -11935.61,E2 -11935.61} C_VEL
LIN {X 0,Y 383.456,Z 706.601,A -85,B 0,C 180,E1 -11936.034,E2 -11936.034} C_VEL
LIN {X 0,Y 387.377,Z 723.254,A -85,B 0,C 180,E1 -11939.262,E2 -11939.262} C_VEL
LIN {X 0,Y 389.043,Z 731.712,A -85,B 0,C 180,E1 -11940.817,E2 -11940.817} C_VEL
LIN {X 0,Y 387.3,Z 752.245,A -85,B 0,C 180,E1 -11944.192,E2 -11944.192} C_VEL
LIN {X 0,Y 385.738,Z 772.501,A -85,B 0,C 180,E1 -11947.514,E2 -11947.514} C_VEL
LIN {X 0,Y 385.023,Z 782.194,A -85,B 0,C 180,E1 -11949.114,E2 -11949.114} C_VEL
LIN {X 0,Y 388.263,Z 810.67,A -85,B 0,C 180,E1 -11949.834,E2 -11949.834} C_VEL
LIN {X 0,Y 389.726,Z 826.884,A -85,B 0,C 180,E1 -11950.218,E2 -11950.218} C_VEL
LIN {X 0,Y 388.719,Z 893.239,A -85,B 0,C 180,E1 -11951.461,E2 -11951.461} C_VEL
LIN {X 0,Y 388.064,Z 906.432,A -85,B 0,C 180,E1 -11951.907,E2 -11951.907} C_VEL
LIN {X 0,Y 387.152,Z 919.724,A -85,B 0,C 180,E1 -11952.579,E2 -11952.579} C_VEL
LIN {X 0,Y 386.205,Z 930.931,A -85,B 0,C 180,E1 -11953.353,E2 -11953.353} C_VEL
LIN {X 0,Y 385.117,Z 942.621,A -85,B 0,C 180,E1 -11954.393,E2 -11954.393} C_VEL
LIN {X 0,Y 384.272,Z 953.207,A -85,B 0,C 180,E1 -11955.579,E2 -11955.579} C_VEL
LIN {X 0,Y 383.713,Z 961.914,A -85,B 0,C 180,E1 -11956.773,E2 -11956.773} C_VEL
LIN {X 0,Y 382.966,Z 969.933,A -85,B 0,C 180,E1 -11958.093,E2 -11958.093} C_VEL
LIN {X 0,Y 382.436,Z 977.817,A -85,B 0,C 180,E1 -11959.686,E2 -11959.686} C_VEL
LIN {X 0,Y 382.223,Z 985.134,A -85,B 0,C 180,E1 -11961.549,E2 -11961.549} C_VEL
LIN {X 0,Y 382.218,Z 990.132,A -85,B 0,C 180,E1 -11963.179,E2 -11963.179} C_VEL
LIN {X 0,Y 382.226,Z 993.78,A -85,B 0,C 180,E1 -11964.732,E2 -11964.732} C_VEL
LIN {X 0,Y 382.369,Z 995.733,A -85,B 0,C 180,E1 -11965.791,E2 -11965.791} C_VEL
LIN {X 0,Y 382.367,Z 997.181,A -85,B 0,C 180,E1 -11966.846,E2 -11966.846} C_VEL
LIN {X 0,Y 382.395,Z 998.217,A -85,B 0,C 180,E1 -11967.901,E2 -11967.901} C_VEL
LIN {X 0,Y 382.438,Z 998.852,A -85,B 0,C 180,E1 -11968.954,E2 -11968.954} C_VEL
LIN {X 0,Y 382.475,Z 999.077,A -85,B 0,C 180,E1 -11970.007,E2 -11970.007} C_VEL
LIN {X 0,Y 382.438,Z 998.842,A -85,B 0,C 180,E1 -11971.06,E2 -11971.06} C_VEL
LIN {X 0,Y 382.396,Z 998.201,A -85,B 0,C 180,E1 -11972.113,E2 -11972.113} C_VEL
LIN {X 0,Y 382.37,Z 997.158,A -85,B 0,C 180,E1 -11973.168,E2 -11973.168} C_VEL
LIN {X 0,Y 382.372,Z 995.7,A -85,B 0,C 180,E1 -11974.223,E2 -11974.223} C_VEL
LIN {X 0,Y 382.185,Z 992.619,A -85,B 0,C 180,E1 -11975.811,E2 -11975.811} C_VEL
LIN {X 0,Y 382.155,Z 988.483,A -85,B 0,C 180,E1 -11977.403,E2 -11977.403} C_VEL
LIN {X 0,Y 382.275,Z 982.144,A -85,B 0,C 180,E1 -11979.264,E2 -11979.264} C_VEL
LIN {X 0,Y 382.612,Z 975.266,A -85,B 0,C 180,E1 -11980.859,E2 -11980.859} C_VEL
LIN {X 0,Y 383.147,Z 966.768,A -85,B 0,C 180,E1 -11982.453,E2 -11982.453} C_VEL
LIN {X 0,Y 383.738,Z 959.938,A -85,B 0,C 180,E1 -11983.51,E2 -11983.51} C_VEL
LIN {X 0,Y 384.521,Z 950.875,A -85,B 0,C 180,E1 -11984.696,E2 -11984.696} C_VEL
LIN {X 0,Y 385.255,Z 941.11,A -85,B 0,C 180,E1 -11985.751,E2 -11985.751} C_VEL
LIN {X 0,Y 386.2,Z 930.676,A -85,B 0,C 180,E1 -11986.661,E2 -11986.661} C_VEL
LIN {X 0,Y 387.218,Z 918.246,A -85,B 0,C 180,E1 -11987.5,E2 -11987.5} C_VEL
LIN {X 0,Y 388.121,Z 905.188,A -85,B 0,C 180,E1 -11988.139,E2 -11988.139} C_VEL
LIN {X 0,Y 388.727,Z 892.487,A -85,B 0,C 180,E1 -11988.553,E2 -11988.553} C_VEL
LIN {X 0,Y 389.542,Z 843.973,A -85,B 0,C 180,E1 -11989.489,E2 -11989.489} C_VEL
LIN {X 0,Y 389.991,Z 822.827,A -85,B 0,C 180,E1 -11990.044,E2 -11990.044} C_VEL
LIN {X 0,Y 387.578,Z 793.272,A -85,B 0,C 180,E1 -11991.074,E2 -11991.074} C_VEL
LIN {X 0,Y 385.433,Z 776.725,A -85,B 0,C 180,E1 -11991.78,E2 -11991.78} C_VEL
LIN {X 0,Y 387.04,Z 755.503,A -85,B 0,C 180,E1 -11995.265,E2 -11995.265} C_VEL
LIN {X 0,Y 388.906,Z 733.267,A -85,B 0,C 180,E1 -11998.914,E2 -11998.914} C_VEL
LIN {X 0,Y 388.72,Z 729.788,A -85,B 0,C 180,E1 -11999.517,E2 -11999.517} C_VEL
LIN {X 0,Y 385.272,Z 714.266,A -85,B 0,C 180,E1 -12002.444,E2 -12002.444} C_VEL
LIN {X 0,Y 382.944,Z 704.785,A -85,B 0,C 180,E1 -12004.323,E2 -12004.323} C_VEL
LIN {X 0,Y 383.004,Z 704.776,A -85,B 0,C 180,E1 -12007.904,E2 -12007.904} C_VEL
LIN {X 0,Y 382.974,Z 704.782,A -85,B 0,C 180,E1 -12011.354,E2 -12011.354} C_VEL
LIN {X 0,Y 382.983,Z 704.776,A -85,B 0,C 180,E1 -12014.301,E2 -12014.301} C_VEL
LIN {X 0,Y 383,Z 704.778,A -85,B 0,C 180,E1 -12017.239,E2 -12017.239} C_VEL
LIN {X 0,Y 383.004,Z 704.774,A -85,B 0,C 180,E1 -12020.422,E2 -12020.422} C_VEL
LIN {X 0,Y 383.031,Z 704.771,A -85,B 0,C 180,E1 -12024.045,E2 -12024.045} C_VEL
LIN {X 0,Y 383.004,Z 704.777,A -85,B 0,C 180,E1 -12027.581,E2 -12027.581} C_VEL
LIN {X 0,Y 382.996,Z 704.777,A -85,B 0,C 180,E1 -12030.3,E2 -12030.3} C_VEL
LIN {X 0,Y 383.024,Z 704.775,A -85,B 0,C 180,E1 -12034.046,E2 -12034.046} C_VEL
LIN {X 0,Y 383.009,Z 704.777,A -85,B 0,C 180,E1 -12037.335,E2 -12037.335} C_VEL
LIN {X 0,Y 383.023,Z 704.776,A -85,B 0,C 180,E1 -12038.159,E2 -12038.159} C_VEL
LIN {X 0,Y 384.05,Z 707.673,A -85,B 0,C 180,E1 -12038.366,E2 -12038.366} C_VEL
LIN {X 0,Y 385.167,Z 709.415,A -85,B 0,C 180,E1 -12038.534,E2 -12038.534} C_VEL
LIN {X 0,Y 391.521,Z 722.145,A -85,B 0,C 180,E1 -12039.529,E2 -12039.529} C_VEL
LIN {X 0,Y 392.812,Z 725.434,A -85,B 0,C 180,E1 -12039.74,E2 -12039.74} C_VEL
LIN {X 0,Y 390.789,Z 785.737,A -85,B 0,C 180,E1 -12041.316,E2 -12041.316} C_VEL
LIN {X 0,Y 390.697,Z 800.329,A -85,B 0,C 180,E1 -12041.821,E2 -12041.821} C_VEL
LIN {X 0,Y 390.288,Z 813.265,A -85,B 0,C 180,E1 -12042.501,E2 -12042.501} C_VEL
LIN {X 0,Y 389.871,Z 822.385,A -85,B 0,C 180,E1 -12043.115,E2 -12043.115} C_VEL
LIN {X 0,Y 389.314,Z 831.954,A -85,B 0,C 180,E1 -12043.911,E2 -12043.911} C_VEL
LIN {X 0,Y 388.618,Z 840.778,A -85,B 0,C 180,E1 -12044.798,E2 -12044.798} C_VEL
LIN {X 0,Y 388.02,Z 849.371,A -85,B 0,C 180,E1 -12045.847,E2 -12045.847} C_VEL
LIN {X 0,Y 387.317,Z 856.64,A -85,B 0,C 180,E1 -12046.89,E2 -12046.89} C_VEL
LIN {X 0,Y 386.749,Z 862.821,A -85,B 0,C 180,E1 -12047.938,E2 -12047.938} C_VEL
LIN {X 0,Y 386.094,Z 869.245,A -85,B 0,C 180,E1 -12049.247,E2 -12049.247} C_VEL
LIN {X 0,Y 385.356,Z 874.594,A -85,B 0,C 180,E1 -12050.553,E2 -12050.553} C_VEL
LIN {X 0,Y 384.815,Z 879.632,A -85,B 0,C 180,E1 -12052.127,E2 -12052.127} C_VEL
LIN {X 0,Y 384.114,Z 883.542,A -85,B 0,C 180,E1 -12053.697,E2 -12053.697} C_VEL
LIN {X 0,Y 383.961,Z 885.572,A -85,B 0,C 180,E1 -12054.749,E2 -12054.749} C_VEL
LIN {X 0,Y 383.555,Z 888.05,A -85,B 0,C 180,E1 -12056.849,E2 -12056.849} C_VEL
LIN {X 0,Y 383.36,Z 888.762,A -85,B 0,C 180,E1 -12057.899,E2 -12057.899} C_VEL
LIN {X 0,Y 383.232,Z 888.935,A -85,B 0,C 180,E1 -12058.949,E2 -12058.949} C_VEL
LIN {X 0,Y 383.128,Z 888.698,A -85,B 0,C 180,E1 -12060,E2 -12060} C_VEL
LIN {X 0,Y 383.12,Z 888.039,A -85,B 0,C 180,E1 -12061.051,E2 -12061.051} C_VEL
LIN {X 0,Y 382.906,Z 885.352,A -85,B 0,C 180,E1 -12063.157,E2 -12063.157} C_VEL
LIN {X 0,Y 383.029,Z 883.443,A -85,B 0,C 180,E1 -12064.209,E2 -12064.209} C_VEL
LIN {X 0,Y 383.42,Z 879.544,A -85,B 0,C 180,E1 -12065.786,E2 -12065.786} C_VEL
LIN {X 0,Y 383.746,Z 873.459,A -85,B 0,C 180,E1 -12067.63,E2 -12067.63} C_VEL
LIN {X 0,Y 383.972,Z 868.071,A -85,B 0,C 180,E1 -12068.95,E2 -12068.95} C_VEL
LIN {X 0,Y 384.353,Z 861.568,A -85,B 0,C 180,E1 -12070.27,E2 -12070.27} C_VEL
LIN {X 0,Y 384.714,Z 855.478,A -85,B 0,C 180,E1 -12071.326,E2 -12071.326} C_VEL
LIN {X 0,Y 385.131,Z 846.309,A -85,B 0,C 180,E1 -12072.649,E2 -12072.649} C_VEL
LIN {X 0,Y 385.556,Z 838.736,A -85,B 0,C 180,E1 -12073.573,E2 -12073.573} C_VEL
LIN {X 0,Y 386.029,Z 829.769,A -85,B 0,C 180,E1 -12074.497,E2 -12074.497} C_VEL
LIN {X 0,Y 386.41,Z 820.344,A -85,B 0,C 180,E1 -12075.308,E2 -12075.308} C_VEL
LIN {X 0,Y 386.777,Z 809.04,A -85,B 0,C 180,E1 -12076.087,E2 -12076.087} C_VEL
LIN {X 0,Y 386.988,Z 798.585,A -85,B 0,C 180,E1 -12076.655,E2 -12076.655} C_VEL
LIN {X 0,Y 387.228,Z 787.963,A -85,B 0,C 180,E1 -12077.085,E2 -12077.085} C_VEL
LIN {X 0,Y 387.405,Z 774.854,A -85,B 0,C 180,E1 -12077.452,E2 -12077.452} C_VEL
LIN {X 0,Y 388.231,Z 720.591,A -85,B 0,C 180,E1 -12078.679,E2 -12078.679} C_VEL
LIN {X 0,Y 383.085,Z 704.766,A -85,B 0,C 180,E1 -12079.283,E2 -12079.283} C_VEL
LIN {X 0,Y 383.009,Z 704.776,A -85,B 0,C 180,E1 -12082.665,E2 -12082.665} C_VEL
LIN {X 0,Y 383.009,Z 704.773,A -85,B 0,C 180,E1 -12086.129,E2 -12086.129} C_VEL
LIN {X 0,Y 382.998,Z 704.774,A -85,B 0,C 180,E1 -12089.7,E2 -12089.7} C_VEL
LIN {X 0,Y 383.019,Z 704.771,A -85,B 0,C 180,E1 -12093.399,E2 -12093.399} C_VEL
LIN {X 0,Y 383.042,Z 704.767,A -85,B 0,C 180,E1 -12096.16,E2 -12096.16} C_VEL
LIN {X 0,Y 383.005,Z 704.772,A -85,B 0,C 180,E1 -12099.579,E2 -12099.579} C_VEL
LIN {X 0,Y 383.026,Z 704.771,A -85,B 0,C 180,E1 -12102.776,E2 -12102.776} C_VEL
LIN {X 0,Y 383.009,Z 704.769,A -85,B 0,C 180,E1 -12105.785,E2 -12105.785} C_VEL
LIN {X 0,Y 382.98,Z 704.776,A -85,B 0,C 180,E1 -12108.798,E2 -12108.798} C_VEL
LIN {X 0,Y 383.01,Z 704.769,A -85,B 0,C 180,E1 -12112.095,E2 -12112.095} C_VEL
LIN {X 0,Y 383.029,Z 704.77,A -85,B 0,C 180,E1 -12115.327,E2 -12115.327} C_VEL
LIN {X 0,Y 382.995,Z 704.775,A -85,B 0,C 180,E1 -12119.077,E2 -12119.077} C_VEL
LIN {X 0,Y 382.98,Z 704.775,A -85,B 0,C 180,E1 -12122.686,E2 -12122.686} C_VEL
LIN {X 0,Y 383.019,Z 704.773,A -85,B 0,C 180,E1 -12126.186,E2 -12126.186} C_VEL
LIN {X 0,Y 383.059,Z 704.772,A -85,B 0,C 180,E1 -12129.537,E2 -12129.537} C_VEL
LIN {X 0,Y 384.631,Z 709.132,A -85,B 0,C 180,E1 -12129.728,E2 -12129.728} C_VEL
LIN {X 0,Y 390.654,Z 723.799,A -85,B 0,C 180,E1 -12130.355,E2 -12130.355} C_VEL
LIN {X 0,Y 390.06,Z 785.265,A -85,B 0,C 180,E1 -12131.515,E2 -12131.515} C_VEL
LIN {X 0,Y 390.041,Z 797.847,A -85,B 0,C 180,E1 -12131.92,E2 -12131.92} C_VEL
LIN {X 0,Y 389.672,Z 810.63,A -85,B 0,C 180,E1 -12132.546,E2 -12132.546} C_VEL
LIN {X 0,Y 389.06,Z 822.524,A -85,B 0,C 180,E1 -12133.339,E2 -12133.339} C_VEL
LIN {X 0,Y 388.412,Z 833.066,A -85,B 0,C 180,E1 -12134.246,E2 -12134.246} C_VEL
LIN {X 0,Y 387.604,Z 843.925,A -85,B 0,C 180,E1 -12135.423,E2 -12135.423} C_VEL
LIN {X 0,Y 386.927,Z 852.7,A -85,B 0,C 180,E1 -12136.603,E2 -12136.603} C_VEL
LIN {X 0,Y 386.146,Z 860.752,A -85,B 0,C 180,E1 -12137.912,E2 -12137.912} C_VEL
LIN {X 0,Y 385.318,Z 868.626,A -85,B 0,C 180,E1 -12139.484,E2 -12139.484} C_VEL
LIN {X 0,Y 384.73,Z 874.296,A -85,B 0,C 180,E1 -12140.888,E2 -12140.888} C_VEL
LIN {X 0,Y 384.269,Z 879.918,A -85,B 0,C 180,E1 -12142.638,E2 -12142.638} C_VEL
LIN {X 0,Y 383.705,Z 883.813,A -85,B 0,C 180,E1 -12144.212,E2 -12144.212} C_VEL
LIN {X 0,Y 383.342,Z 886.68,A -85,B 0,C 180,E1 -12145.788,E2 -12145.788} C_VEL
LIN {X 0,Y 383.294,Z 888.04,A -85,B 0,C 180,E1 -12146.84,E2 -12146.84} C_VEL
LIN {X 0,Y 383.291,Z 889.002,A -85,B 0,C 180,E1 -12147.892,E2 -12147.892} C_VEL
LIN {X 0,Y 383.147,Z 889.845,A -85,B 0,C 180,E1 -12149.993,E2 -12149.993} C_VEL
LIN {X 0,Y 383.308,Z 889.085,A -85,B 0,C 180,E1 -12152.094,E2 -12152.094} C_VEL
LIN {X 0,Y 383.305,Z 887.212,A -85,B 0,C 180,E1 -12153.911,E2 -12153.911} C_VEL
LIN {X 0,Y 382.683,Z 886.52,A -85,B 0,C 180,E1 -12154.494,E2 -12154.494} C_VEL
LIN {X 0,Y 377.491,Z 883.946,A -85,B 0,C 180,E1 -12156.336,E2 -12156.336} C_VEL
LIN {X 0,Y 377.152,Z 882.698,A -85,B 0,C 180,E1 -12156.907,E2 -12156.907} C_VEL
LIN {X 0,Y 377.719,Z 876.928,A -85,B 0,C 180,E1 -12158.906,E2 -12158.906} C_VEL
LIN {X 0,Y 378.203,Z 871.263,A -85,B 0,C 180,E1 -12160.43,E2 -12160.43} C_VEL
LIN {X 0,Y 379.095,Z 863.82,A -85,B 0,C 180,E1 -12162.03,E2 -12162.03} C_VEL
LIN {X 0,Y 379.94,Z 856.187,A -85,B 0,C 180,E1 -12163.361,E2 -12163.361} C_VEL
LIN {X 0,Y 380.67,Z 846.874,A -85,B 0,C 180,E1 -12164.697,E2 -12164.697} C_VEL
LIN {X 0,Y 381.526,Z 836.501,A -85,B 0,C 180,E1 -12165.895,E2 -12165.895} C_VEL
LIN {X 0,Y 382.367,Z 824.866,A -85,B 0,C 180,E1 -12166.957,E2 -12166.957} C_VEL
LIN {X 0,Y 383.019,Z 812.398,A -85,B 0,C 180,E1 -12167.821,E2 -12167.821} C_VEL
LIN {X 0,Y 383.332,Z 799.917,A -85,B 0,C 180,E1 -12168.463,E2 -12168.463} C_VEL
LIN {X 0,Y 383.473,Z 788.138,A -85,B 0,C 180,E1 -12168.871,E2 -12168.871} C_VEL
LIN {X 0,Y 383.655,Z 754.696,A -85,B 0,C 180,E1 -12169.537,E2 -12169.537} C_VEL
LIN {X 0,Y 384.044,Z 725.432,A -85,B 0,C 180,E1 -12170.089,E2 -12170.089} C_VEL
LIN {X 0,Y 376.025,Z 706.122,A -85,B 0,C 180,E1 -12170.949,E2 -12170.949} C_VEL
LIN {X 0,Y 375.956,Z 705.656,A -85,B 0,C 180,E1 -12170.993,E2 -12170.993} C_VEL
LIN {X 0,Y 375.971,Z 705.648,A -85,B 0,C 180,E1 -12174.273,E2 -12174.273} C_VEL
LIN {X 0,Y 375.995,Z 705.644,A -85,B 0,C 180,E1 -12176.644,E2 -12176.644} C_VEL
LIN {X 0,Y 375.936,Z 705.652,A -85,B 0,C 180,E1 -12180.305,E2 -12180.305} C_VEL
LIN {X 0,Y 375.927,Z 705.654,A -85,B 0,C 180,E1 -12184.104,E2 -12184.104} C_VEL
LIN {X 0,Y 375.919,Z 705.657,A -85,B 0,C 180,E1 -12186.733,E2 -12186.733} C_VEL
LIN {X 0,Y 375.959,Z 705.654,A -85,B 0,C 180,E1 -12189.965,E2 -12189.965} C_VEL
LIN {X 0,Y 375.957,Z 705.644,A -85,B 0,C 180,E1 -12193.748,E2 -12193.748} C_VEL
LIN {X 0,Y 375.952,Z 705.646,A -85,B 0,C 180,E1 -12196.793,E2 -12196.793} C_VEL
LIN {X 0,Y 375.949,Z 705.654,A -85,B 0,C 180,E1 -12200.021,E2 -12200.021} C_VEL
LIN {X 0,Y 375.911,Z 705.66,A -85,B 0,C 180,E1 -12203.489,E2 -12203.489} C_VEL
LIN {X 0,Y 375.905,Z 705.656,A -85,B 0,C 180,E1 -12205.883,E2 -12205.883} C_VEL
LIN {X 0,Y 375.91,Z 705.658,A -85,B 0,C 180,E1 -12209.682,E2 -12209.682} C_VEL
LIN {X 0,Y 375.935,Z 705.653,A -85,B 0,C 180,E1 -12212.136,E2 -12212.136} C_VEL
LIN {X 0,Y 375.943,Z 705.653,A -85,B 0,C 180,E1 -12214.534,E2 -12214.534} C_VEL
LIN {X 0,Y 375.901,Z 705.657,A -85,B 0,C 180,E1 -12218.042,E2 -12218.042} C_VEL
LIN {X 0,Y 375.94,Z 705.648,A -85,B 0,C 180,E1 -12221.47,E2 -12221.47} C_VEL
LIN {X 0,Y 375.993,Z 705.651,A -85,B 0,C 180,E1 -12224.83,E2 -12224.83} C_VEL
LIN {X 0,Y 375.99,Z 705.647,A -85,B 0,C 180,E1 -12228.135,E2 -12228.135} C_VEL
LIN {X 0,Y 376.149,Z 705.629,A -85,B 0,C 180,E1 -12231.916,E2 -12231.916} C_VEL
LIN {X 0,Y 376.107,Z 705.635,A -85,B 0,C 180,E1 -12234.639,E2 -12234.639} C_VEL
LIN {X 0,Y 376.286,Z 705.611,A -85,B 0,C 180,E1 -12237.859,E2 -12237.859} C_VEL
LIN {X 0,Y 376.418,Z 705.597,A -85,B 0,C 180,E1 -12240,E2 -12240} C_VEL
LIN {X 0,Y 376.149,Z 705.625,A -85,B 0,C 180,E1 -12243.213,E2 -12243.213} C_VEL
LIN {X 0,Y 376.176,Z 705.627,A -85,B 0,C 180,E1 -12246.436,E2 -12246.436} C_VEL
LIN {X 0,Y 376.053,Z 705.637,A -85,B 0,C 180,E1 -12249.683,E2 -12249.683} C_VEL
LIN {X 0,Y 376.02,Z 705.647,A -85,B 0,C 180,E1 -12253.66,E2 -12253.66} C_VEL
LIN {X 0,Y 375.982,Z 705.651,A -85,B 0,C 180,E1 -12257.402,E2 -12257.402} C_VEL
LIN {X 0,Y 375.912,Z 705.649,A -85,B 0,C 180,E1 -12260.836,E2 -12260.836} C_VEL
LIN {X 0,Y 375.929,Z 705.653,A -85,B 0,C 180,E1 -12264.286,E2 -12264.286} C_VEL
LIN {X 0,Y 375.957,Z 705.647,A -85,B 0,C 180,E1 -12266.657,E2 -12266.657} C_VEL
LIN {X 0,Y 375.916,Z 705.655,A -85,B 0,C 180,E1 -12269.084,E2 -12269.084} C_VEL
LIN {X 0,Y 375.899,Z 705.658,A -85,B 0,C 180,E1 -12272.834,E2 -12272.834} C_VEL
LIN {X 0,Y 375.903,Z 705.658,A -85,B 0,C 180,E1 -12275.422,E2 -12275.422} C_VEL
LIN {X 0,Y 375.925,Z 705.644,A -85,B 0,C 180,E1 -12278.277,E2 -12278.277} C_VEL
LIN {X 0,Y 375.941,Z 705.656,A -85,B 0,C 180,E1 -12281.617,E2 -12281.617} C_VEL
LIN {X 0,Y 375.971,Z 705.65,A -85,B 0,C 180,E1 -12285.262,E2 -12285.262} C_VEL
LIN {X 0,Y 375.959,Z 705.655,A -85,B 0,C 180,E1 -12289.148,E2 -12289.148} C_VEL
LIN {X 0,Y 375.93,Z 705.658,A -85,B 0,C 180,E1 -12291.92,E2 -12291.92} C_VEL
LIN {X 0,Y 375.965,Z 705.784,A -85,B 0,C 180,E1 -12295.302,E2 -12295.302} C_VEL
LIN {X 0,Y 379.657,Z 721.111,A -85,B 0,C 180,E1 -12298.378,E2 -12298.378} C_VEL
LIN {X 0,Y 382.056,Z 732.459,A -85,B 0,C 180,E1 -12300.533,E2 -12300.533} C_VEL
LIN {X 0,Y 381.146,Z 744.463,A -85,B 0,C 180,E1 -12302.56,E2 -12302.56} C_VEL
LIN {X 0,Y 379.284,Z 766.458,A -85,B 0,C 180,E1 -12306.242,E2 -12306.242} C_VEL
LIN {X 0,Y 378.103,Z 781.158,A -85,B 0,C 180,E1 -12308.713,E2 -12308.713} C_VEL
LIN {X 0,Y 381.744,Z 813.179,A -85,B 0,C 180,E1 -12309.542,E2 -12309.542} C_VEL
LIN {X 0,Y 383.023,Z 827.855,A -85,B 0,C 180,E1 -12309.896,E2 -12309.896} C_VEL
LIN {X 0,Y 381.959,Z 892.233,A -85,B 0,C 180,E1 -12311.121,E2 -12311.121} C_VEL
LIN {X 0,Y 381.339,Z 905.43,A -85,B 0,C 180,E1 -12311.576,E2 -12311.576} C_VEL
LIN {X 0,Y 380.351,Z 918.712,A -85,B 0,C 180,E1 -12312.258,E2 -12312.258} C_VEL
LIN {X 0,Y 379.387,Z 929.919,A -85,B 0,C 180,E1 -12313.045,E2 -12313.045} C_VEL
LIN {X 0,Y 378.21,Z 941.601,A -85,B 0,C 180,E1 -12314.101,E2 -12314.101} C_VEL
LIN {X 0,Y 377.373,Z 952.197,A -85,B 0,C 180,E1 -12315.31,E2 -12315.31} C_VEL
LIN {X 0,Y 376.811,Z 959.062,A -85,B 0,C 180,E1 -12316.251,E2 -12316.251} C_VEL
LIN {X 0,Y 375.951,Z 968.912,A -85,B 0,C 180,E1 -12317.868,E2 -12317.868} C_VEL
LIN {X 0,Y 375.396,Z 976.797,A -85,B 0,C 180,E1 -12319.491,E2 -12319.491} C_VEL
LIN {X 0,Y 375.149,Z 984.115,A -85,B 0,C 180,E1 -12321.388,E2 -12321.388} C_VEL
LIN {X 0,Y 375.148,Z 989.441,A -85,B 0,C 180,E1 -12323.169,E2 -12323.169} C_VEL
LIN {X 0,Y 375.156,Z 992.768,A -85,B 0,C 180,E1 -12324.633,E2 -12324.633} C_VEL
LIN {X 0,Y 375.3,Z 994.722,A -85,B 0,C 180,E1 -12325.712,E2 -12325.712} C_VEL
LIN {X 0,Y 375.322,Z 996.175,A -85,B 0,C 180,E1 -12326.787,E2 -12326.787} C_VEL
LIN {X 0,Y 375.355,Z 997.212,A -85,B 0,C 180,E1 -12327.861,E2 -12327.861} C_VEL
LIN {X 0,Y 375.403,Z 997.848,A -85,B 0,C 180,E1 -12328.934,E2 -12328.934} C_VEL
LIN {X 0,Y 375.446,Z 998.074,A -85,B 0,C 180,E1 -12330.007,E2 -12330.007} C_VEL
LIN {X 0,Y 375.404,Z 997.838,A -85,B 0,C 180,E1 -12331.08,E2 -12331.08} C_VEL
LIN {X 0,Y 375.356,Z 997.195,A -85,B 0,C 180,E1 -12332.153,E2 -12332.153} C_VEL
LIN {X 0,Y 375.325,Z 996.151,A -85,B 0,C 180,E1 -12333.227,E2 -12333.227} C_VEL
LIN {X 0,Y 375.303,Z 994.688,A -85,B 0,C 180,E1 -12334.303,E2 -12334.303} C_VEL
LIN {X 0,Y 375.13,Z 991.606,A -85,B 0,C 180,E1 -12335.921,E2 -12335.921} C_VEL
LIN {X 0,Y 375.109,Z 987.468,A -85,B 0,C 180,E1 -12337.543,E2 -12337.543} C_VEL
LIN {X 0,Y 375.227,Z 981.124,A -85,B 0,C 180,E1 -12339.439,E2 -12339.439} C_VEL
LIN {X 0,Y 375.591,Z 974.244,A -85,B 0,C 180,E1 -12341.064,E2 -12341.064} C_VEL
LIN {X 0,Y 376.169,Z 965.746,A -85,B 0,C 180,E1 -12342.688,E2 -12342.688} C_VEL
LIN {X 0,Y 376.679,Z 959.526,A -85,B 0,C 180,E1 -12343.674,E2 -12343.674} C_VEL
LIN {X 0,Y 377.699,Z 948.759,A -85,B 0,C 180,E1 -12345.106,E2 -12345.106} C_VEL
LIN {X 0,Y 378.506,Z 938.744,A -85,B 0,C 180,E1 -12346.178,E2 -12346.178} C_VEL
LIN {X 0,Y 379.694,Z 926.151,A -85,B 0,C 180,E1 -12347.233,E2 -12347.233} C_VEL
LIN {X 0,Y 380.729,Z 913.818,A -85,B 0,C 180,E1 -12348.017,E2 -12348.017} C_VEL
LIN {X 0,Y 381.54,Z 900.819,A -85,B 0,C 180,E1 -12348.602,E2 -12348.602} C_VEL
LIN {X 0,Y 382.073,Z 886.993,A -85,B 0,C 180,E1 -12348.993,E2 -12348.993} C_VEL
LIN {X 0,Y 382.619,Z 858.998,A -85,B 0,C 180,E1 -12349.546,E2 -12349.546} C_VEL
LIN {X 0,Y 383.604,Z 824.004,A -85,B 0,C 180,E1 -12350.47,E2 -12350.47} C_VEL
LIN {X 0,Y 381.308,Z 794.316,A -85,B 0,C 180,E1 -12351.552,E2 -12351.552} C_VEL
LIN {X 0,Y 378.636,Z 774.321,A -85,B 0,C 180,E1 -12352.429,E2 -12352.429} C_VEL
LIN {X 0,Y 380.392,Z 752.813,A -85,B 0,C 180,E1 -12356.033,E2 -12356.033} C_VEL
LIN {X 0,Y 382.058,Z 734.025,A -85,B 0,C 180,E1 -12359.18,E2 -12359.18} C_VEL
LIN {X 0,Y 381.273,Z 728.701,A -85,B 0,C 180,E1 -12360.157,E2 -12360.157} C_VEL
LIN {X 0,Y 378.113,Z 714.485,A -85,B 0,C 180,E1 -12362.912,E2 -12362.912} C_VEL
LIN {X 0,Y 375.924,Z 705.652,A -85,B 0,C 180,E1 -12364.721,E2 -12364.721} C_VEL
LIN {X 0,Y 375.946,Z 705.655,A -85,B 0,C 180,E1 -12368.265,E2 -12368.265} C_VEL
LIN {X 0,Y 375.927,Z 705.658,A -85,B 0,C 180,E1 -12371.599,E2 -12371.599} C_VEL
LIN {X 0,Y 375.922,Z 705.66,A -85,B 0,C 180,E1 -12375.275,E2 -12375.275} C_VEL
LIN {X 0,Y 375.932,Z 705.655,A -85,B 0,C 180,E1 -12378.406,E2 -12378.406} C_VEL
LIN {X 0,Y 375.971,Z 705.652,A -85,B 0,C 180,E1 -12381.912,E2 -12381.912} C_VEL
LIN {X 0,Y 375.994,Z 705.651,A -85,B 0,C 180,E1 -12385.336,E2 -12385.336} C_VEL
LIN {X 0,Y 375.957,Z 705.652,A -85,B 0,C 180,E1 -12388.438,E2 -12388.438} C_VEL
LIN {X 0,Y 375.971,Z 705.653,A -85,B 0,C 180,E1 -12391.478,E2 -12391.478} C_VEL
LIN {X 0,Y 375.957,Z 705.655,A -85,B 0,C 180,E1 -12394.535,E2 -12394.535} C_VEL
LIN {X 0,Y 375.983,Z 705.799,A -85,B 0,C 180,E1 -12397.45,E2 -12397.45} C_VEL
LIN {X 0,Y 377.071,Z 708.62,A -85,B 0,C 180,E1 -12397.672,E2 -12397.672} C_VEL
LIN {X 0,Y 378.492,Z 711.057,A -85,B 0,C 180,E1 -12397.916,E2 -12397.916} C_VEL
LIN {X 0,Y 384.716,Z 722.921,A -85,B 0,C 180,E1 -12398.937,E2 -12398.937} C_VEL
LIN {X 0,Y 386.631,Z 727.54,A -85,B 0,C 180,E1 -12399.27,E2 -12399.27} C_VEL
LIN {X 0,Y 384.454,Z 786.54,A -85,B 0,C 180,E1 -12400.858,E2 -12400.858} C_VEL
LIN {X 0,Y 384.329,Z 801.003,A -85,B 0,C 180,E1 -12401.371,E2 -12401.371} C_VEL
LIN {X 0,Y 383.884,Z 814.449,A -85,B 0,C 180,E1 -12402.087,E2 -12402.087} C_VEL
LIN {X 0,Y 383.415,Z 823.794,A -85,B 0,C 180,E1 -12402.726,E2 -12402.726} C_VEL
LIN {X 0,Y 382.787,Z 834.026,A -85,B 0,C 180,E1 -12403.603,E2 -12403.603} C_VEL
LIN {X 0,Y 382.05,Z 842.937,A -85,B 0,C 180,E1 -12404.53,E2 -12404.53} C_VEL
LIN {X 0,Y 381.389,Z 851.346,A -85,B 0,C 180,E1 -12405.595,E2 -12405.595} C_VEL
LIN {X 0,Y 380.623,Z 858.46,A -85,B 0,C 180,E1 -12406.655,E2 -12406.655} C_VEL
LIN {X 0,Y 379.995,Z 864.51,A -85,B 0,C 180,E1 -12407.72,E2 -12407.72} C_VEL
LIN {X 0,Y 379.223,Z 871.465,A -85,B 0,C 180,E1 -12409.199,E2 -12409.199} C_VEL
LIN {X 0,Y 378.523,Z 876.14,A -85,B 0,C 180,E1 -12410.381,E2 -12410.381} C_VEL
LIN {X 0,Y 377.956,Z 881.106,A -85,B 0,C 180,E1 -12411.983,E2 -12411.983} C_VEL
LIN {X 0,Y 377.488,Z 883.865,A -85,B 0,C 180,E1 -12413.049,E2 -12413.049} C_VEL
LIN {X 0,Y 377.018,Z 886.902,A -85,B 0,C 180,E1 -12414.652,E2 -12414.652} C_VEL
LIN {X 0,Y 376.791,Z 888.277,A -85,B 0,C 180,E1 -12415.721,E2 -12415.721} C_VEL
LIN {X 0,Y 376.377,Z 889.927,A -85,B 0,C 180,E1 -12417.86,E2 -12417.86} C_VEL
LIN {X 0,Y 376.24,Z 890.053,A -85,B 0,C 180,E1 -12418.93,E2 -12418.93} C_VEL
LIN {X 0,Y 376.111,Z 889.774,A -85,B 0,C 180,E1 -12420,E2 -12420} C_VEL
LIN {X 0,Y 376.098,Z 889.049,A -85,B 0,C 180,E1 -12421.071,E2 -12421.071} C_VEL
LIN {X 0,Y 375.979,Z 887.845,A -85,B 0,C 180,E1 -12422.143,E2 -12422.143} C_VEL
LIN {X 0,Y 375.995,Z 884.254,A -85,B 0,C 180,E1 -12424.288,E2 -12424.288} C_VEL
LIN {X 0,Y 376.393,Z 880.234,A -85,B 0,C 180,E1 -12425.895,E2 -12425.895} C_VEL
LIN {X 0,Y 376.644,Z 875.048,A -85,B 0,C 180,E1 -12427.505,E2 -12427.505} C_VEL
LIN {X 0,Y 376.972,Z 868.764,A -85,B 0,C 180,E1 -12429.064,E2 -12429.064} C_VEL
LIN {X 0,Y 377.291,Z 863.354,A -85,B 0,C 180,E1 -12430.193,E2 -12430.193} C_VEL
LIN {X 0,Y 377.738,Z 855.648,A -85,B 0,C 180,E1 -12431.538,E2 -12431.538} C_VEL
LIN {X 0,Y 378.141,Z 847.342,A -85,B 0,C 180,E1 -12432.751,E2 -12432.751} C_VEL
LIN {X 0,Y 378.639,Z 838.539,A -85,B 0,C 180,E1 -12433.826,E2 -12433.826} C_VEL
LIN {X 0,Y 379.092,Z 829.333,A -85,B 0,C 180,E1 -12434.768,E2 -12434.768} C_VEL
LIN {X 0,Y 379.467,Z 820.905,A -85,B 0,C 180,E1 -12435.495,E2 -12435.495} C_VEL
LIN {X 0,Y 379.813,Z 810.144,A -85,B 0,C 180,E1 -12436.253,E2 -12436.253} C_VEL
LIN {X 0,Y 380.052,Z 799.779,A -85,B 0,C 180,E1 -12436.829,E2 -12436.829} C_VEL
LIN {X 0,Y 380.278,Z 789.333,A -85,B 0,C 180,E1 -12437.269,E2 -12437.269} C_VEL
LIN {X 0,Y 380.426,Z 776.482,A -85,B 0,C 180,E1 -12437.643,E2 -12437.643} C_VEL
LIN {X 0,Y 381.321,Z 721.969,A -85,B 0,C 180,E1 -12438.91,E2 -12438.91} C_VEL
LIN {X 0,Y 376.048,Z 705.641,A -85,B 0,C 180,E1 -12439.53,E2 -12439.53} C_VEL
LIN {X 0,Y 375.995,Z 705.646,A -85,B 0,C 180,E1 -12443.658,E2 -12443.658} C_VEL
LIN {X 0,Y 375.944,Z 705.657,A -85,B 0,C 180,E1 -12446.658,E2 -12446.658} C_VEL
LIN {X 0,Y 375.937,Z 705.658,A -85,B 0,C 180,E1 -12449.082,E2 -12449.082} C_VEL
LIN {X 0,Y 375.958,Z 705.652,A -85,B 0,C 180,E1 -12451.562,E2 -12451.562} C_VEL
LIN {X 0,Y 375.995,Z 705.648,A -85,B 0,C 180,E1 -12454.664,E2 -12454.664} C_VEL
LIN {X 0,Y 375.955,Z 705.651,A -85,B 0,C 180,E1 -12458.26,E2 -12458.26} C_VEL
LIN {X 0,Y 375.933,Z 705.652,A -85,B 0,C 180,E1 -12461.594,E2 -12461.594} C_VEL
LIN {X 0,Y 375.94,Z 705.652,A -85,B 0,C 180,E1 -12464.727,E2 -12464.727} C_VEL
LIN {X 0,Y 375.926,Z 705.652,A -85,B 0,C 180,E1 -12467.693,E2 -12467.693} C_VEL
LIN {X 0,Y 375.952,Z 705.649,A -85,B 0,C 180,E1 -12470.53,E2 -12470.53} C_VEL
LIN {X 0,Y 375.975,Z 705.648,A -85,B 0,C 180,E1 -12473.494,E2 -12473.494} C_VEL
LIN {X 0,Y 375.975,Z 705.646,A -85,B 0,C 180,E1 -12475.884,E2 -12475.884} C_VEL
LIN {X 0,Y 375.976,Z 705.648,A -85,B 0,C 180,E1 -12479.683,E2 -12479.683} C_VEL
LIN {X 0,Y 375.932,Z 705.652,A -85,B 0,C 180,E1 -12482.13,E2 -12482.13} C_VEL
LIN {X 0,Y 375.95,Z 705.652,A -85,B 0,C 180,E1 -12484.529,E2 -12484.529} C_VEL
LIN {X 0,Y 375.982,Z 705.651,A -85,B 0,C 180,E1 -12486.881,E2 -12486.881} C_VEL
LIN {X 0,Y 375.974,Z 705.654,A -85,B 0,C 180,E1 -12489.127,E2 -12489.127} C_VEL
LIN {X 0,Y 377.672,Z 710.148,A -85,B 0,C 180,E1 -12489.336,E2 -12489.336} C_VEL
LIN {X 0,Y 384.131,Z 725.939,A -85,B 0,C 180,E1 -12490.029,E2 -12490.029} C_VEL
LIN {X 0,Y 383.375,Z 783.744,A -85,B 0,C 180,E1 -12491.122,E2 -12491.122} C_VEL
LIN {X 0,Y 383.361,Z 797.186,A -85,B 0,C 180,E1 -12491.529,E2 -12491.529} C_VEL
LIN {X 0,Y 383.046,Z 809.352,A -85,B 0,C 180,E1 -12492.096,E2 -12492.096} C_VEL
LIN {X 0,Y 382.462,Z 821.668,A -85,B 0,C 180,E1 -12492.896,E2 -12492.896} C_VEL
LIN {X 0,Y 381.767,Z 833.039,A -85,B 0,C 180,E1 -12493.864,E2 -12493.864} C_VEL
LIN {X 0,Y 381.011,Z 842.715,A -85,B 0,C 180,E1 -12494.891,E2 -12494.891} C_VEL
LIN {X 0,Y 380.244,Z 851.917,A -85,B 0,C 180,E1 -12496.091,E2 -12496.091} C_VEL
LIN {X 0,Y 379.458,Z 860.297,A -85,B 0,C 180,E1 -12497.424,E2 -12497.424} C_VEL
LIN {X 0,Y 378.526,Z 868.432,A -85,B 0,C 180,E1 -12499.023,E2 -12499.023} C_VEL
LIN {X 0,Y 377.793,Z 875.299,A -85,B 0,C 180,E1 -12500.719,E2 -12500.719} C_VEL
LIN {X 0,Y 377.303,Z 880.921,A -85,B 0,C 180,E1 -12502.501,E2 -12502.501} C_VEL
LIN {X 0,Y 376.715,Z 884.817,A -85,B 0,C 180,E1 -12504.104,E2 -12504.104} C_VEL
LIN {X 0,Y 376.333,Z 887.683,A -85,B 0,C 180,E1 -12505.709,E2 -12505.709} C_VEL
LIN {X 0,Y 376.278,Z 889.043,A -85,B 0,C 180,E1 -12506.781,E2 -12506.781} C_VEL
LIN {X 0,Y 376.273,Z 890.004,A -85,B 0,C 180,E1 -12507.852,E2 -12507.852} C_VEL
LIN {X 0,Y 376.121,Z 890.847,A -85,B 0,C 180,E1 -12509.993,E2 -12509.993} C_VEL
LIN {X 0,Y 376.287,Z 890.087,A -85,B 0,C 180,E1 -12512.133,E2 -12512.133} C_VEL
LIN {X 0,Y 376.319,Z 887.857,A -85,B 0,C 180,E1 -12514.277,E2 -12514.277} C_VEL
LIN {X 0,Y 376.705,Z 885.046,A -85,B 0,C 180,E1 -12515.882,E2 -12515.882} C_VEL
LIN {X 0,Y 377.152,Z 882.698,A -85,B 0,C 180,E1 -12516.907,E2 -12516.907} C_VEL
LIN {X 0,Y 376.945,Z 880.656,A -85,B 0,C 180,E1 -12517.745,E2 -12517.745} C_VEL
LIN {X 0,Y 375.643,Z 878.561,A -85,B 0,C 180,E1 -12518.568,E2 -12518.568} C_VEL
LIN {X 0,Y 371.963,Z 872.865,A -85,B 0,C 180,E1 -12520.435,E2 -12520.435} C_VEL
LIN {X 0,Y 371.633,Z 869.763,A -85,B 0,C 180,E1 -12521.211,E2 -12521.211} C_VEL
LIN {X 0,Y 372.567,Z 861.921,A -85,B 0,C 180,E1 -12522.798,E2 -12522.798} C_VEL
LIN {X 0,Y 373.389,Z 853.706,A -85,B 0,C 180,E1 -12524.155,E2 -12524.155} C_VEL
LIN {X 0,Y 374.255,Z 843.545,A -85,B 0,C 180,E1 -12525.513,E2 -12525.513} C_VEL
LIN {X 0,Y 375.19,Z 833.083,A -85,B 0,C 180,E1 -12526.626,E2 -12526.626} C_VEL
LIN {X 0,Y 375.934,Z 821.3,A -85,B 0,C 180,E1 -12527.623,E2 -12527.623} C_VEL
LIN {X 0,Y 376.448,Z 808.778,A -85,B 0,C 180,E1 -12528.418,E2 -12528.418} C_VEL
LIN {X 0,Y 376.677,Z 795.662,A -85,B 0,C 180,E1 -12529.013,E2 -12529.013} C_VEL
LIN {X 0,Y 376.795,Z 783.139,A -85,B 0,C 180,E1 -12529.36,E2 -12529.36} C_VEL
LIN {X 0,Y 377.419,Z 733.669,A -85,B 0,C 180,E1 -12530.312,E2 -12530.312} C_VEL
LIN {X 0,Y 377.282,Z 726.781,A -85,B 0,C 180,E1 -12530.458,E2 -12530.458} C_VEL
LIN {X 0,Y 369.608,Z 708.82,A -85,B 0,C 180,E1 -12531.294,E2 -12531.294} C_VEL
LIN {X 0,Y 368.888,Z 706.533,A -85,B 0,C 180,E1 -12531.414,E2 -12531.414} C_VEL
LIN {X 0,Y 368.934,Z 706.525,A -85,B 0,C 180,E1 -12534.767,E2 -12534.767} C_VEL
LIN {X 0,Y 368.938,Z 706.526,A -85,B 0,C 180,E1 -12537.195,E2 -12537.195} C_VEL
LIN {X 0,Y 368.9,Z 706.532,A -85,B 0,C 180,E1 -12540.945,E2 -12540.945} C_VEL
LIN {X 0,Y 368.895,Z 706.532,A -85,B 0,C 180,E1 -12544.993,E2 -12544.993} C_VEL
LIN {X 0,Y 368.874,Z 706.519,A -85,B 0,C 180,E1 -12548.633,E2 -12548.633} C_VEL
LIN {X 0,Y 368.9,Z 706.535,A -85,B 0,C 180,E1 -12552.012,E2 -12552.012} C_VEL
LIN {X 0,Y 368.946,Z 706.509,A -85,B 0,C 180,E1 -12555.186,E2 -12555.186} C_VEL
LIN {X 0,Y 368.893,Z 706.536,A -85,B 0,C 180,E1 -12558.179,E2 -12558.179} C_VEL
LIN {X 0,Y 368.862,Z 706.534,A -85,B 0,C 180,E1 -12561.352,E2 -12561.352} C_VEL
LIN {X 0,Y 368.881,Z 706.53,A -85,B 0,C 180,E1 -12565.14,E2 -12565.14} C_VEL
LIN {X 0,Y 368.871,Z 706.533,A -85,B 0,C 180,E1 -12569.041,E2 -12569.041} C_VEL
LIN {X 0,Y 368.92,Z 706.521,A -85,B 0,C 180,E1 -12571.559,E2 -12571.559} C_VEL
LIN {X 0,Y 368.937,Z 706.529,A -85,B 0,C 180,E1 -12574.015,E2 -12574.015} C_VEL
LIN {X 0,Y 368.869,Z 706.529,A -85,B 0,C 180,E1 -12577.601,E2 -12577.601} C_VEL
LIN {X 0,Y 368.89,Z 706.527,A -85,B 0,C 180,E1 -12581.102,E2 -12581.102} C_VEL
LIN {X 0,Y 368.932,Z 706.527,A -85,B 0,C 180,E1 -12584.532,E2 -12584.532} C_VEL
LIN {X 0,Y 368.944,Z 706.523,A -85,B 0,C 180,E1 -12587.905,E2 -12587.905} C_VEL
LIN {X 0,Y 369.118,Z 706.504,A -85,B 0,C 180,E1 -12591.843,E2 -12591.843} C_VEL
LIN {X 0,Y 369.079,Z 706.512,A -85,B 0,C 180,E1 -12594.537,E2 -12594.537} C_VEL
LIN {X 0,Y 369.252,Z 706.487,A -85,B 0,C 180,E1 -12597.818,E2 -12597.818} C_VEL
LIN {X 0,Y 369.388,Z 706.473,A -85,B 0,C 180,E1 -12600,E2 -12600} C_VEL
LIN {X 0,Y 369.087,Z 706.505,A -85,B 0,C 180,E1 -12603.275,E2 -12603.275} C_VEL
LIN {X 0,Y 369.135,Z 706.505,A -85,B 0,C 180,E1 -12606.559,E2 -12606.559} C_VEL
LIN {X 0,Y 369.052,Z 706.509,A -85,B 0,C 180,E1 -12608.763,E2 -12608.763} C_VEL
LIN {X 0,Y 368.944,Z 706.526,A -85,B 0,C 180,E1 -12612.095,E2 -12612.095} C_VEL
LIN {X 0,Y 368.932,Z 706.532,A -85,B 0,C 180,E1 -12615.468,E2 -12615.468} C_VEL
LIN {X 0,Y 368.89,Z 706.532,A -85,B 0,C 180,E1 -12618.898,E2 -12618.898} C_VEL
LIN {X 0,Y 368.866,Z 706.534,A -85,B 0,C 180,E1 -12622.399,E2 -12622.399} C_VEL
LIN {X 0,Y 368.937,Z 706.522,A -85,B 0,C 180,E1 -12625.985,E2 -12625.985} C_VEL
LIN {X 0,Y 368.907,Z 706.528,A -85,B 0,C 180,E1 -12628.818,E2 -12628.818} C_VEL
LIN {X 0,Y 368.852,Z 706.539,A -85,B 0,C 180,E1 -12632.243,E2 -12632.243} C_VEL
LIN {X 0,Y 368.873,Z 706.533,A -85,B 0,C 180,E1 -12635.007,E2 -12635.007} C_VEL
LIN {X 0,Y 368.861,Z 706.522,A -85,B 0,C 180,E1 -12638.648,E2 -12638.648} C_VEL
LIN {X 0,Y 368.894,Z 706.536,A -85,B 0,C 180,E1 -12642.027,E2 -12642.027} C_VEL
LIN {X 0,Y 368.946,Z 706.526,A -85,B 0,C 180,E1 -12645.2,E2 -12645.2} C_VEL
LIN {X 0,Y 368.899,Z 706.527,A -85,B 0,C 180,E1 -12648.193,E2 -12648.193} C_VEL
LIN {X 0,Y 368.874,Z 706.534,A -85,B 0,C 180,E1 -12651.367,E2 -12651.367} C_VEL
LIN {X 0,Y 368.9,Z 706.685,A -85,B 0,C 180,E1 -12654.905,E2 -12654.905} C_VEL
LIN {X 0,Y 371.905,Z 718.852,A -85,B 0,C 180,E1 -12657.425,E2 -12657.425} C_VEL
LIN {X 0,Y 375.078,Z 733.197,A -85,B 0,C 180,E1 -12660.239,E2 -12660.239} C_VEL
LIN {X 0,Y 374.938,Z 738.551,A -85,B 0,C 180,E1 -12661.181,E2 -12661.181} C_VEL
LIN {X 0,Y 372.708,Z 762.615,A -85,B 0,C 180,E1 -12665.293,E2 -12665.293} C_VEL
LIN {X 0,Y 371.291,Z 779.968,A -85,B 0,C 180,E1 -12668.275,E2 -12668.275} C_VEL
LIN {X 0,Y 375,Z 813.258,A -85,B 0,C 180,E1 -12669.179,E2 -12669.179} C_VEL
LIN {X 0,Y 376.335,Z 829.236,A -85,B 0,C 180,E1 -12669.57,E2 -12669.57} C_VEL
LIN {X 0,Y 375.219,Z 891.229,A -85,B 0,C 180,E1 -12670.768,E2 -12670.768} C_VEL
LIN {X 0,Y 374.602,Z 904.425,A -85,B 0,C 180,E1 -12671.233,E2 -12671.233} C_VEL
LIN {X 0,Y 373.593,Z 917.705,A -85,B 0,C 180,E1 -12671.926,E2 -12671.926} C_VEL
LIN {X 0,Y 372.564,Z 928.905,A -85,B 0,C 180,E1 -12672.725,E2 -12672.725} C_VEL
LIN {X 0,Y 371.396,Z 940.593,A -85,B 0,C 180,E1 -12673.801,E2 -12673.801} C_VEL
LIN {X 0,Y 370.58,Z 950.091,A -85,B 0,C 180,E1 -12674.893,E2 -12674.893} C_VEL
LIN {X 0,Y 369.762,Z 958.776,A -85,B 0,C 180,E1 -12676.098,E2 -12676.098} C_VEL
LIN {X 0,Y 368.928,Z 967.889,A -85,B 0,C 180,E1 -12677.633,E2 -12677.633} C_VEL
LIN {X 0,Y 368.351,Z 975.776,A -85,B 0,C 180,E1 -12679.287,E2 -12679.287} C_VEL
LIN {X 0,Y 368.071,Z 983.095,A -85,B 0,C 180,E1 -12681.221,E2 -12681.221} C_VEL
LIN {X 0,Y 368.074,Z 988.736,A -85,B 0,C 180,E1 -12683.163,E2 -12683.163} C_VEL
LIN {X 0,Y 368.089,Z 991.756,A -85,B 0,C 180,E1 -12684.53,E2 -12684.53} C_VEL
LIN {X 0,Y 368.234,Z 993.712,A -85,B 0,C 180,E1 -12685.629,E2 -12685.629} C_VEL
LIN {X 0,Y 368.277,Z 995.168,A -85,B 0,C 180,E1 -12686.725,E2 -12686.725} C_VEL
LIN {X 0,Y 368.314,Z 996.207,A -85,B 0,C 180,E1 -12687.82,E2 -12687.82} C_VEL
LIN {X 0,Y 368.369,Z 996.844,A -85,B 0,C 180,E1 -12688.914,E2 -12688.914} C_VEL
LIN {X 0,Y 368.416,Z 997.071,A -85,B 0,C 180,E1 -12690.007,E2 -12690.007} C_VEL
LIN {X 0,Y 368.369,Z 996.834,A -85,B 0,C 180,E1 -12691.1,E2 -12691.1} C_VEL
LIN {X 0,Y 368.315,Z 996.19,A -85,B 0,C 180,E1 -12692.194,E2 -12692.194} C_VEL
LIN {X 0,Y 368.28,Z 995.144,A -85,B 0,C 180,E1 -12693.289,E2 -12693.289} C_VEL
LIN {X 0,Y 368.236,Z 993.676,A -85,B 0,C 180,E1 -12694.385,E2 -12694.385} C_VEL
LIN {X 0,Y 368.072,Z 990.593,A -85,B 0,C 180,E1 -12696.035,E2 -12696.035} C_VEL
LIN {X 0,Y 368.056,Z 986.452,A -85,B 0,C 180,E1 -12697.688,E2 -12697.688} C_VEL
LIN {X 0,Y 368.166,Z 980.101,A -85,B 0,C 180,E1 -12699.622,E2 -12699.622} C_VEL
LIN {X 0,Y 368.545,Z 973.217,A -85,B 0,C 180,E1 -12701.278,E2 -12701.278} C_VEL
LIN {X 0,Y 369.212,Z 964.726,A -85,B 0,C 180,E1 -12702.931,E2 -12702.931} C_VEL
LIN {X 0,Y 369.988,Z 955.643,A -85,B 0,C 180,E1 -12704.36,E2 -12704.36} C_VEL
LIN {X 0,Y 370.799,Z 946.553,A -85,B 0,C 180,E1 -12705.535,E2 -12705.535} C_VEL
LIN {X 0,Y 371.863,Z 936.29,A -85,B 0,C 180,E1 -12706.616,E2 -12706.616} C_VEL
LIN {X 0,Y 372.904,Z 925.13,A -85,B 0,C 180,E1 -12707.557,E2 -12707.557} C_VEL
LIN {X 0,Y 373.948,Z 912.793,A -85,B 0,C 180,E1 -12708.355,E2 -12708.355} C_VEL
LIN {X 0,Y 374.808,Z 899.795,A -85,B 0,C 180,E1 -12708.949,E2 -12708.949} C_VEL
LIN {X 0,Y 375.36,Z 886.005,A -85,B 0,C 180,E1 -12709.346,E2 -12709.346} C_VEL
LIN {X 0,Y 375.844,Z 867.722,A -85,B 0,C 180,E1 -12709.782,E2 -12709.782} C_VEL
LIN {X 0,Y 377.322,Z 825.315,A -85,B 0,C 180,E1 -12710.923,E2 -12710.923} C_VEL
LIN {X 0,Y 375.136,Z 795.354,A -85,B 0,C 180,E1 -12712.056,E2 -12712.056} C_VEL
LIN {X 0,Y 372.291,Z 774.799,A -85,B 0,C 180,E1 -12713.006,E2 -12713.006} C_VEL
LIN {X 0,Y 371.878,Z 771.417,A -85,B 0,C 180,E1 -12713.19,E2 -12713.19} C_VEL
LIN {X 0,Y 373.679,Z 751.828,A -85,B 0,C 180,E1 -12716.537,E2 -12716.537} C_VEL
LIN {X 0,Y 375.178,Z 734.805,A -85,B 0,C 180,E1 -12719.453,E2 -12719.453} C_VEL
LIN {X 0,Y 372.91,Z 723.262,A -85,B 0,C 180,E1 -12721.68,E2 -12721.68} C_VEL
LIN {X 0,Y 369.458,Z 708.843,A -85,B 0,C 180,E1 -12724.622,E2 -12724.622} C_VEL
LIN {X 0,Y 368.881,Z 706.523,A -85,B 0,C 180,E1 -12725.137,E2 -12725.137} C_VEL
LIN {X 0,Y 368.889,Z 706.533,A -85,B 0,C 180,E1 -12728.636,E2 -12728.636} C_VEL
LIN {X 0,Y 368.872,Z 706.535,A -85,B 0,C 180,E1 -12732.008,E2 -12732.008} C_VEL
LIN {X 0,Y 368.874,Z 706.536,A -85,B 0,C 180,E1 -12735.175,E2 -12735.175} C_VEL
LIN {X 0,Y 368.879,Z 706.534,A -85,B 0,C 180,E1 -12738.177,E2 -12738.177} C_VEL
LIN {X 0,Y 368.895,Z 706.535,A -85,B 0,C 180,E1 -12741.369,E2 -12741.369} C_VEL
LIN {X 0,Y 368.95,Z 706.527,A -85,B 0,C 180,E1 -12745.148,E2 -12745.148} C_VEL
LIN {X 0,Y 368.917,Z 706.533,A -85,B 0,C 180,E1 -12749.045,E2 -12749.045} C_VEL
LIN {X 0,Y 368.931,Z 706.53,A -85,B 0,C 180,E1 -12751.56,E2 -12751.56} C_VEL
LIN {X 0,Y 368.935,Z 706.53,A -85,B 0,C 180,E1 -12755.223,E2 -12755.223} C_VEL
LIN {X 0,Y 368.97,Z 706.604,A -85,B 0,C 180,E1 -12756.664,E2 -12756.664} C_VEL
LIN {X 0,Y 369.963,Z 709.397,A -85,B 0,C 180,E1 -12756.897,E2 -12756.897} C_VEL
LIN {X 0,Y 371.324,Z 711.462,A -85,B 0,C 180,E1 -12757.132,E2 -12757.132} C_VEL
LIN {X 0,Y 377.855,Z 723.714,A -85,B 0,C 180,E1 -12758.292,E2 -12758.292} C_VEL
LIN {X 0,Y 380.492,Z 729.303,A -85,B 0,C 180,E1 -12758.74,E2 -12758.74} C_VEL
LIN {X 0,Y 378.19,Z 786.895,A -85,B 0,C 180,E1 -12760.363,E2 -12760.363} C_VEL
LIN {X 0,Y 378.064,Z 800.394,A -85,B 0,C 180,E1 -12760.839,E2 -12760.839} C_VEL
LIN {X 0,Y 377.681,Z 813.354,A -85,B 0,C 180,E1 -12761.488,E2 -12761.488} C_VEL
LIN {X 0,Y 377.029,Z 825.236,A -85,B 0,C 180,E1 -12762.312,E2 -12762.312} C_VEL
LIN {X 0,Y 376.362,Z 835.087,A -85,B 0,C 180,E1 -12763.176,E2 -12763.176} C_VEL
LIN {X 0,Y 375.583,Z 843.976,A -85,B 0,C 180,E1 -12764.117,E2 -12764.117} C_VEL
LIN {X 0,Y 374.96,Z 851.49,A -85,B 0,C 180,E1 -12765.065,E2 -12765.065} C_VEL
LIN {X 0,Y 374.175,Z 858.79,A -85,B 0,C 180,E1 -12766.144,E2 -12766.144} C_VEL
LIN {X 0,Y 373.289,Z 866.332,A -85,B 0,C 180,E1 -12767.496,E2 -12767.496} C_VEL
LIN {X 0,Y 372.577,Z 872.325,A -85,B 0,C 180,E1 -12768.797,E2 -12768.797} C_VEL
LIN {X 0,Y 371.698,Z 877.708,A -85,B 0,C 180,E1 -12770.202,E2 -12770.202} C_VEL
LIN {X 0,Y 371.279,Z 881.186,A -85,B 0,C 180,E1 -12771.29,E2 -12771.29} C_VEL
LIN {X 0,Y 370.585,Z 885.288,A -85,B 0,C 180,E1 -12772.919,E2 -12772.919} C_VEL
LIN {X 0,Y 370.076,Z 888.241,A -85,B 0,C 180,E1 -12774.551,E2 -12774.551} C_VEL
LIN {X 0,Y 369.845,Z 889.602,A -85,B 0,C 180,E1 -12775.641,E2 -12775.641} C_VEL
LIN {X 0,Y 369.391,Z 891.106,A -85,B 0,C 180,E1 -12777.819,E2 -12777.819} C_VEL
LIN {X 0,Y 369.246,Z 891.181,A -85,B 0,C 180,E1 -12778.909,E2 -12778.909} C_VEL
LIN {X 0,Y 369.094,Z 890.852,A -85,B 0,C 180,E1 -12780,E2 -12780} C_VEL
LIN {X 0,Y 369.075,Z 890.036,A -85,B 0,C 180,E1 -12781.091,E2 -12781.091} C_VEL
LIN {X 0,Y 368.954,Z 888.808,A -85,B 0,C 180,E1 -12782.183,E2 -12782.183} C_VEL
LIN {X 0,Y 368.962,Z 885.05,A -85,B 0,C 180,E1 -12784.37,E2 -12784.37} C_VEL
LIN {X 0,Y 369.368,Z 880.921,A -85,B 0,C 180,E1 -12786.007,E2 -12786.007} C_VEL
LIN {X 0,Y 369.625,Z 875.616,A -85,B 0,C 180,E1 -12787.649,E2 -12787.649} C_VEL
LIN {X 0,Y 369.895,Z 870.868,A -85,B 0,C 180,E1 -12788.864,E2 -12788.864} C_VEL
LIN {X 0,Y 370.297,Z 863.641,A -85,B 0,C 180,E1 -12790.388,E2 -12790.388} C_VEL
LIN {X 0,Y 370.677,Z 857.513,A -85,B 0,C 180,E1 -12791.483,E2 -12791.483} C_VEL
LIN {X 0,Y 371.137,Z 848.302,A -85,B 0,C 180,E1 -12792.856,E2 -12792.856} C_VEL
LIN {X 0,Y 371.633,Z 839.464,A -85,B 0,C 180,E1 -12793.953,E2 -12793.953} C_VEL
LIN {X 0,Y 372.107,Z 830.222,A -85,B 0,C 180,E1 -12794.912,E2 -12794.912} C_VEL
LIN {X 0,Y 372.513,Z 821.202,A -85,B 0,C 180,E1 -12795.695,E2 -12795.695} C_VEL
LIN {X 0,Y 372.862,Z 810.951,A -85,B 0,C 180,E1 -12796.423,E2 -12796.423} C_VEL
LIN {X 0,Y 373.098,Z 800.532,A -85,B 0,C 180,E1 -12797.011,E2 -12797.011} C_VEL
LIN {X 0,Y 373.321,Z 790.016,A -85,B 0,C 180,E1 -12797.46,E2 -12797.46} C_VEL
LIN {X 0,Y 373.464,Z 777.202,A -85,B 0,C 180,E1 -12797.842,E2 -12797.842} C_VEL
LIN {X 0,Y 374.405,Z 723.234,A -85,B 0,C 180,E1 -12799.137,E2 -12799.137} C_VEL
LIN {X 0,Y 368.961,Z 706.524,A -85,B 0,C 180,E1 -12799.79,E2 -12799.79} C_VEL
LIN {X 0,Y 368.968,Z 706.522,A -85,B 0,C 180,E1 -12803.579,E2 -12803.579} C_VEL
LIN {X 0,Y 368.888,Z 706.532,A -85,B 0,C 180,E1 -12807.21,E2 -12807.21} C_VEL
LIN {X 0,Y 368.915,Z 706.528,A -85,B 0,C 180,E1 -12809.691,E2 -12809.691} C_VEL
LIN {X 0,Y 368.916,Z 706.53,A -85,B 0,C 180,E1 -12813.041,E2 -12813.041} C_VEL
LIN {X 0,Y 368.931,Z 706.525,A -85,B 0,C 180,E1 -12816.195,E2 -12816.195} C_VEL
LIN {X 0,Y 368.894,Z 706.533,A -85,B 0,C 180,E1 -12818.955,E2 -12818.955} C_VEL
LIN {X 0,Y 368.878,Z 706.529,A -85,B 0,C 180,E1 -12822.002,E2 -12822.002} C_VEL
LIN {X 0,Y 368.893,Z 706.532,A -85,B 0,C 180,E1 -12825.172,E2 -12825.172} C_VEL
LIN {X 0,Y 368.879,Z 706.529,A -85,B 0,C 180,E1 -12828.171,E2 -12828.171} C_VEL
LIN {X 0,Y 368.894,Z 706.53,A -85,B 0,C 180,E1 -12831.363,E2 -12831.363} C_VEL
LIN {X 0,Y 368.948,Z 706.523,A -85,B 0,C 180,E1 -12835.142,E2 -12835.142} C_VEL
LIN {X 0,Y 368.914,Z 706.528,A -85,B 0,C 180,E1 -12839.039,E2 -12839.039} C_VEL
LIN {X 0,Y 368.923,Z 706.528,A -85,B 0,C 180,E1 -12841.553,E2 -12841.553} C_VEL
LIN {X 0,Y 368.934,Z 706.526,A -85,B 0,C 180,E1 -12844.009,E2 -12844.009} C_VEL
LIN {X 0,Y 368.908,Z 706.534,A -85,B 0,C 180,E1 -12847.597,E2 -12847.597} C_VEL
LIN {X 0,Y 368.956,Z 706.527,A -85,B 0,C 180,E1 -12848.693,E2 -12848.693} C_VEL
LIN {X 0,Y 370.472,Z 710.75,A -85,B 0,C 180,E1 -12848.905,E2 -12848.905} C_VEL
LIN {X 0,Y 377.354,Z 727.086,A -85,B 0,C 180,E1 -12849.657,E2 -12849.657} C_VEL
LIN {X 0,Y 376.725,Z 786.628,A -85,B 0,C 180,E1 -12850.82,E2 -12850.82} C_VEL
LIN {X 0,Y 376.659,Z 800.039,A -85,B 0,C 180,E1 -12851.261,E2 -12851.261} C_VEL
LIN {X 0,Y 376.278,Z 812.653,A -85,B 0,C 180,E1 -12851.904,E2 -12851.904} C_VEL
LIN {X 0,Y 375.616,Z 824.541,A -85,B 0,C 180,E1 -12852.724,E2 -12852.724} C_VEL
LIN {X 0,Y 374.904,Z 835.082,A -85,B 0,C 180,E1 -12853.662,E2 -12853.662} C_VEL
LIN {X 0,Y 374.019,Z 845.938,A -85,B 0,C 180,E1 -12854.881,E2 -12854.881} C_VEL
LIN {X 0,Y 373.268,Z 854.712,A -85,B 0,C 180,E1 -12856.104,E2 -12856.104} C_VEL
LIN {X 0,Y 372.417,Z 862.762,A -85,B 0,C 180,E1 -12857.459,E2 -12857.459} C_VEL
LIN {X 0,Y 371.507,Z 870.636,A -85,B 0,C 180,E1 -12859.089,E2 -12859.089} C_VEL
LIN {X 0,Y 370.859,Z 876.302,A -85,B 0,C 180,E1 -12860.543,E2 -12860.543} C_VEL
LIN {X 0,Y 370.339,Z 881.925,A -85,B 0,C 180,E1 -12862.36,E2 -12862.36} C_VEL
LIN {X 0,Y 369.726,Z 885.82,A -85,B 0,C 180,E1 -12863.992,E2 -12863.992} C_VEL
LIN {X 0,Y 369.325,Z 888.687,A -85,B 0,C 180,E1 -12865.628,E2 -12865.628} C_VEL
LIN {X 0,Y 369.261,Z 890.047,A -85,B 0,C 180,E1 -12866.72,E2 -12866.72} C_VEL
LIN {X 0,Y 369.254,Z 891.006,A -85,B 0,C 180,E1 -12867.811,E2 -12867.811} C_VEL
LIN {X 0,Y 369.095,Z 891.85,A -85,B 0,C 180,E1 -12869.993,E2 -12869.993} C_VEL
LIN {X 0,Y 369.266,Z 891.089,A -85,B 0,C 180,E1 -12872.174,E2 -12872.174} C_VEL
LIN {X 0,Y 369.31,Z 888.859,A -85,B 0,C 180,E1 -12874.358,E2 -12874.358} C_VEL
LIN {X 0,Y 369.716,Z 886.047,A -85,B 0,C 180,E1 -12875.994,E2 -12875.994} C_VEL
LIN {X 0,Y 370.308,Z 882.225,A -85,B 0,C 180,E1 -12877.627,E2 -12877.627} C_VEL
LIN {X 0,Y 370.834,Z 876.754,A -85,B 0,C 180,E1 -12879.433,E2 -12879.433} C_VEL
LIN {X 0,Y 371.633,Z 869.763,A -85,B 0,C 180,E1 -12881.211,E2 -12881.211} C_VEL
LIN {X 0,Y 371.403,Z 866.454,A -85,B 0,C 180,E1 -12881.966,E2 -12881.966} C_VEL
LIN {X 0,Y 369.284,Z 860.896,A -85,B 0,C 180,E1 -12883.198,E2 -12883.198} C_VEL
LIN {X 0,Y 367.174,Z 854.796,A -85,B 0,C 180,E1 -12884.371,E2 -12884.371} C_VEL
LIN {X 0,Y 366.949,Z 850.599,A -85,B 0,C 180,E1 -12885.021,E2 -12885.021} C_VEL
LIN {X 0,Y 367.802,Z 841.038,A -85,B 0,C 180,E1 -12886.219,E2 -12886.219} C_VEL
LIN {X 0,Y 368.765,Z 829.61,A -85,B 0,C 180,E1 -12887.354,E2 -12887.354} C_VEL
LIN {X 0,Y 369.538,Z 817.347,A -85,B 0,C 180,E1 -12888.301,E2 -12888.301} C_VEL
LIN {X 0,Y 369.889,Z 804.924,A -85,B 0,C 180,E1 -12889.016,E2 -12889.016} C_VEL
LIN {X 0,Y 370.101,Z 792.4,A -85,B 0,C 180,E1 -12889.508,E2 -12889.508} C_VEL
LIN {X 0,Y 370.186,Z 767.243,A -85,B 0,C 180,E1 -12890.063,E2 -12890.063} C_VEL
LIN {X 0,Y 370.811,Z 728.928,A -85,B 0,C 180,E1 -12890.807,E2 -12890.807} C_VEL
LIN {X 0,Y 362.595,Z 709.734,A -85,B 0,C 180,E1 -12891.73,E2 -12891.73} C_VEL
LIN {X 0,Y 361.889,Z 707.401,A -85,B 0,C 180,E1 -12891.848,E2 -12891.848} C_VEL
LIN {X 0,Y 361.905,Z 707.402,A -85,B 0,C 180,E1 -12895.282,E2 -12895.282} C_VEL
LIN {X 0,Y 361.882,Z 707.402,A -85,B 0,C 180,E1 -12897.771,E2 -12897.771} C_VEL
LIN {X 0,Y 361.808,Z 707.418,A -85,B 0,C 180,E1 -12901.621,E2 -12901.621} C_VEL
LIN {X 0,Y 361.84,Z 707.414,A -85,B 0,C 180,E1 -12905.337,E2 -12905.337} C_VEL
LIN {X 0,Y 361.836,Z 707.398,A -85,B 0,C 180,E1 -12909.02,E2 -12909.02} C_VEL
LIN {X 0,Y 361.845,Z 707.412,A -85,B 0,C 180,E1 -12912.433,E2 -12912.433} C_VEL
LIN {X 0,Y 361.884,Z 707.392,A -85,B 0,C 180,E1 -12915.921,E2 -12915.921} C_VEL
LIN {X 0,Y 361.857,Z 707.412,A -85,B 0,C 180,E1 -12919.225,E2 -12919.225} C_VEL
LIN {X 0,Y 361.816,Z 707.413,A -85,B 0,C 180,E1 -12922.976,E2 -12922.976} C_VEL
LIN {X 0,Y 361.806,Z 707.412,A -85,B 0,C 180,E1 -12926.624,E2 -12926.624} C_VEL
LIN {X 0,Y 361.817,Z 707.414,A -85,B 0,C 180,E1 -12929.667,E2 -12929.667} C_VEL
LIN {X 0,Y 361.892,Z 707.403,A -85,B 0,C 180,E1 -12933.47,E2 -12933.47} C_VEL
LIN {X 0,Y 361.827,Z 707.406,A -85,B 0,C 180,E1 -12937.14,E2 -12937.14} C_VEL
LIN {X 0,Y 361.839,Z 707.409,A -85,B 0,C 180,E1 -12940.719,E2 -12940.719} C_VEL
LIN {X 0,Y 361.866,Z 707.401,A -85,B 0,C 180,E1 -12943.063,E2 -12943.063} C_VEL
LIN {X 0,Y 361.931,Z 707.405,A -85,B 0,C 180,E1 -12946.525,E2 -12946.525} C_VEL
LIN {X 0,Y 361.966,Z 707.386,A -85,B 0,C 180,E1 -12949.936,E2 -12949.936} C_VEL
LIN {X 0,Y 362.096,Z 707.381,A -85,B 0,C 180,E1 -12953.312,E2 -12953.312} C_VEL
LIN {X 0,Y 362.218,Z 707.364,A -85,B 0,C 180,E1 -12957.776,E2 -12957.776} C_VEL
LIN {X 0,Y 362.358,Z 707.348,A -85,B 0,C 180,E1 -12960,E2 -12960} C_VEL
LIN {X 0,Y 362.218,Z 707.359,A -85,B 0,C 180,E1 -12962.224,E2 -12962.224} C_VEL
LIN {X 0,Y 362.096,Z 707.383,A -85,B 0,C 180,E1 -12966.688,E2 -12966.688} C_VEL
LIN {X 0,Y 361.966,Z 707.391,A -85,B 0,C 180,E1 -12970.064,E2 -12970.064} C_VEL
LIN {X 0,Y 361.929,Z 707.4,A -85,B 0,C 180,E1 -12973.901,E2 -12973.901} C_VEL
LIN {X 0,Y 361.901,Z 707.405,A -85,B 0,C 180,E1 -12977.942,E2 -12977.942} C_VEL
LIN {X 0,Y 361.818,Z 707.408,A -85,B 0,C 180,E1 -12981.658,E2 -12981.658} C_VEL
LIN {X 0,Y 361.865,Z 707.405,A -85,B 0,C 180,E1 -12985.295,E2 -12985.295} C_VEL
LIN {X 0,Y 361.861,Z 707.409,A -85,B 0,C 180,E1 -12987.783,E2 -12987.783} C_VEL
LIN {X 0,Y 361.801,Z 707.414,A -85,B 0,C 180,E1 -12991.633,E2 -12991.633} C_VEL
LIN {X 0,Y 361.819,Z 707.412,A -85,B 0,C 180,E1 -12995.351,E2 -12995.351} C_VEL
LIN {X 0,Y 361.823,Z 707.398,A -85,B 0,C 180,E1 -12999.034,E2 -12999.034} C_VEL
LIN {X 0,Y 361.839,Z 707.412,A -85,B 0,C 180,E1 -13002.448,E2 -13002.448} C_VEL
LIN {X 0,Y 361.886,Z 707.408,A -85,B 0,C 180,E1 -13005.936,E2 -13005.936} C_VEL
LIN {X 0,Y 361.865,Z 707.411,A -85,B 0,C 180,E1 -13009.239,E2 -13009.239} C_VEL
LIN {X 0,Y 361.837,Z 707.409,A -85,B 0,C 180,E1 -13012.991,E2 -13012.991} C_VEL
LIN {X 0,Y 361.86,Z 707.474,A -85,B 0,C 180,E1 -13014.47,E2 -13014.47} C_VEL
LIN {X 0,Y 364.852,Z 719.649,A -85,B 0,C 180,E1 -13017.056,E2 -13017.056} C_VEL
LIN {X 0,Y 368.123,Z 734.377,A -85,B 0,C 180,E1 -13020.015,E2 -13020.015} C_VEL
LIN {X 0,Y 368.112,Z 739.122,A -85,B 0,C 180,E1 -13020.877,E2 -13020.877} C_VEL
LIN {X 0,Y 365.821,Z 762.777,A -85,B 0,C 180,E1 -13025.008,E2 -13025.008} C_VEL
LIN {X 0,Y 364.429,Z 779.261,A -85,B 0,C 180,E1 -13027.877,E2 -13027.877} C_VEL
LIN {X 0,Y 368.409,Z 814.734,A -85,B 0,C 180,E1 -13028.839,E2 -13028.839} C_VEL
LIN {X 0,Y 369.652,Z 829.219,A -85,B 0,C 180,E1 -13029.203,E2 -13029.203} C_VEL
LIN {X 0,Y 368.481,Z 890.223,A -85,B 0,C 180,E1 -13030.402,E2 -13030.402} C_VEL
LIN {X 0,Y 367.871,Z 903.418,A -85,B 0,C 180,E1 -13030.876,E2 -13030.876} C_VEL
LIN {X 0,Y 366.861,Z 916.7,A -85,B 0,C 180,E1 -13031.582,E2 -13031.582} C_VEL
LIN {X 0,Y 365.755,Z 927.891,A -85,B 0,C 180,E1 -13032.393,E2 -13032.393} C_VEL
LIN {X 0,Y 364.533,Z 939.576,A -85,B 0,C 180,E1 -13033.487,E2 -13033.487} C_VEL
LIN {X 0,Y 363.658,Z 949.071,A -85,B 0,C 180,E1 -13034.598,E2 -13034.598} C_VEL
LIN {X 0,Y 362.73,Z 957.547,A -85,B 0,C 180,E1 -13035.792,E2 -13035.792} C_VEL
LIN {X 0,Y 362.26,Z 963.833,A -85,B 0,C 180,E1 -13036.832,E2 -13036.832} C_VEL
LIN {X 0,Y 361.519,Z 972.298,A -85,B 0,C 180,E1 -13038.515,E2 -13038.515} C_VEL
LIN {X 0,Y 361.11,Z 979.163,A -85,B 0,C 180,E1 -13040.203,E2 -13040.203} C_VEL
LIN {X 0,Y 360.989,Z 985.492,A -85,B 0,C 180,E1 -13042.175,E2 -13042.175} C_VEL
LIN {X 0,Y 361.037,Z 989.629,A -85,B 0,C 180,E1 -13043.862,E2 -13043.862} C_VEL
LIN {X 0,Y 361.17,Z 992.701,A -85,B 0,C 180,E1 -13045.544,E2 -13045.544} C_VEL
LIN {X 0,Y 361.232,Z 994.162,A -85,B 0,C 180,E1 -13046.662,E2 -13046.662} C_VEL
LIN {X 0,Y 361.273,Z 995.202,A -85,B 0,C 180,E1 -13047.778,E2 -13047.778} C_VEL
LIN {X 0,Y 361.334,Z 995.841,A -85,B 0,C 180,E1 -13048.893,E2 -13048.893} C_VEL
LIN {X 0,Y 361.387,Z 996.068,A -85,B 0,C 180,E1 -13050.007,E2 -13050.007} C_VEL
LIN {X 0,Y 361.334,Z 995.83,A -85,B 0,C 180,E1 -13051.122,E2 -13051.122} C_VEL
LIN {X 0,Y 361.274,Z 995.184,A -85,B 0,C 180,E1 -13052.237,E2 -13052.237} C_VEL
LIN {X 0,Y 361.235,Z 994.136,A -85,B 0,C 180,E1 -13053.353,E2 -13053.353} C_VEL
LIN {X 0,Y 361.172,Z 992.665,A -85,B 0,C 180,E1 -13054.471,E2 -13054.471} C_VEL
LIN {X 0,Y 361.016,Z 989.58,A -85,B 0,C 180,E1 -13056.153,E2 -13056.153} C_VEL
LIN {X 0,Y 360.998,Z 985.435,A -85,B 0,C 180,E1 -13057.839,E2 -13057.839} C_VEL
LIN {X 0,Y 361.117,Z 979.079,A -85,B 0,C 180,E1 -13059.812,E2 -13059.812} C_VEL
LIN {X 0,Y 361.53,Z 972.195,A -85,B 0,C 180,E1 -13061.5,E2 -13061.5} C_VEL
LIN {X 0,Y 362.267,Z 963.707,A -85,B 0,C 180,E1 -13063.183,E2 -13063.183} C_VEL
LIN {X 0,Y 362.801,Z 956.641,A -85,B 0,C 180,E1 -13064.339,E2 -13064.339} C_VEL
LIN {X 0,Y 363.736,Z 947.793,A -85,B 0,C 180,E1 -13065.557,E2 -13065.557} C_VEL
LIN {X 0,Y 364.705,Z 938.046,A -85,B 0,C 180,E1 -13066.664,E2 -13066.664} C_VEL
LIN {X 0,Y 365.735,Z 927.607,A -85,B 0,C 180,E1 -13067.623,E2 -13067.623} C_VEL
LIN {X 0,Y 366.956,Z 915.187,A -85,B 0,C 180,E1 -13068.5,E2 -13068.5} C_VEL
LIN {X 0,Y 367.888,Z 902.116,A -85,B 0,C 180,E1 -13069.175,E2 -13069.175} C_VEL
LIN {X 0,Y 369.058,Z 879.546,A -85,B 0,C 180,E1 -13069.943,E2 -13069.943} C_VEL
LIN {X 0,Y 371.059,Z 826.239,A -85,B 0,C 180,E1 -13071.413,E2 -13071.413} C_VEL
LIN {X 0,Y 369.09,Z 797.176,A -85,B 0,C 180,E1 -13072.554,E2 -13072.554} C_VEL
LIN {X 0,Y 366.392,Z 776.538,A -85,B 0,C 180,E1 -13073.554,E2 -13073.554} C_VEL
LIN {X 0,Y 365.275,Z 768.456,A -85,B 0,C 180,E1 -13073.988,E2 -13073.988} C_VEL
LIN {X 0,Y 367.397,Z 745.814,A -85,B 0,C 180,E1 -13077.943,E2 -13077.943} C_VEL
LIN {X 0,Y 368.219,Z 737.224,A -85,B 0,C 180,E1 -13079.444,E2 -13079.444} C_VEL
LIN {X 0,Y 367.752,Z 732.958,A -85,B 0,C 180,E1 -13080.25,E2 -13080.25} C_VEL
LIN {X 0,Y 364.837,Z 719.518,A -85,B 0,C 180,E1 -13082.955,E2 -13082.955} C_VEL
LIN {X 0,Y 361.84,Z 707.398,A -85,B 0,C 180,E1 -13085.543,E2 -13085.543} C_VEL
LIN {X 0,Y 361.84,Z 707.412,A -85,B 0,C 180,E1 -13089.02,E2 -13089.02} C_VEL
LIN {X 0,Y 361.832,Z 707.411,A -85,B 0,C 180,E1 -13092.836,E2 -13092.836} C_VEL
LIN {X 0,Y 361.823,Z 707.413,A -85,B 0,C 180,E1 -13095.952,E2 -13095.952} C_VEL
LIN {X 0,Y 361.83,Z 707.414,A -85,B 0,C 180,E1 -13099.252,E2 -13099.252} C_VEL
LIN {X 0,Y 361.88,Z 707.406,A -85,B 0,C 180,E1 -13102.983,E2 -13102.983} C_VEL
LIN {X 0,Y 361.878,Z 707.405,A -85,B 0,C 180,E1 -13106.634,E2 -13106.634} C_VEL
LIN {X 0,Y 361.868,Z 707.409,A -85,B 0,C 180,E1 -13109.671,E2 -13109.671} C_VEL
LIN {X 0,Y 361.882,Z 707.408,A -85,B 0,C 180,E1 -13113.469,E2 -13113.469} C_VEL
LIN {X 0,Y 361.916,Z 707.552,A -85,B 0,C 180,E1 -13115.796,E2 -13115.796} C_VEL
LIN {X 0,Y 362.942,Z 710.332,A -85,B 0,C 180,E1 -13116.043,E2 -13116.043} C_VEL
LIN {X 0,Y 364.394,Z 712.248,A -85,B 0,C 180,E1 -13116.307,E2 -13116.307} C_VEL
LIN {X 0,Y 371.102,Z 724.539,A -85,B 0,C 180,E1 -13117.589,E2 -13117.589} C_VEL
LIN {X 0,Y 374.504,Z 731.842,A -85,B 0,C 180,E1 -13118.226,E2 -13118.226} C_VEL
LIN {X 0,Y 372.013,Z 787.301,A -85,B 0,C 180,E1 -13119.832,E2 -13119.832} C_VEL
LIN {X 0,Y 371.837,Z 800.53,A -85,B 0,C 180,E1 -13120.308,E2 -13120.308} C_VEL
LIN {X 0,Y 371.489,Z 811.556,A -85,B 0,C 180,E1 -13120.853,E2 -13120.853} C_VEL
LIN {X 0,Y 370.806,Z 825.162,A -85,B 0,C 180,E1 -13121.748,E2 -13121.748} C_VEL
LIN {X 0,Y 369.992,Z 836.343,A -85,B 0,C 180,E1 -13122.735,E2 -13122.735} C_VEL
LIN {X 0,Y 369.173,Z 845.235,A -85,B 0,C 180,E1 -13123.692,E2 -13123.692} C_VEL
LIN {X 0,Y 368.379,Z 853.639,A -85,B 0,C 180,E1 -13124.792,E2 -13124.792} C_VEL
LIN {X 0,Y 367.544,Z 860.744,A -85,B 0,C 180,E1 -13125.889,E2 -13125.889} C_VEL
LIN {X 0,Y 366.799,Z 866.828,A -85,B 0,C 180,E1 -13126.989,E2 -13126.989} C_VEL
LIN {X 0,Y 365.966,Z 873.187,A -85,B 0,C 180,E1 -13128.368,E2 -13128.368} C_VEL
LIN {X 0,Y 365.301,Z 877.534,A -85,B 0,C 180,E1 -13129.469,E2 -13129.469} C_VEL
LIN {X 0,Y 364.451,Z 882.752,A -85,B 0,C 180,E1 -13131.126,E2 -13131.126} C_VEL
LIN {X 0,Y 363.698,Z 886.723,A -85,B 0,C 180,E1 -13132.784,E2 -13132.784} C_VEL
LIN {X 0,Y 363.133,Z 889.574,A -85,B 0,C 180,E1 -13134.447,E2 -13134.447} C_VEL
LIN {X 0,Y 362.895,Z 890.926,A -85,B 0,C 180,E1 -13135.557,E2 -13135.557} C_VEL
LIN {X 0,Y 362.403,Z 892.29,A -85,B 0,C 180,E1 -13137.777,E2 -13137.777} C_VEL
LIN {X 0,Y 362.249,Z 892.313,A -85,B 0,C 180,E1 -13138.888,E2 -13138.888} C_VEL
LIN {X 0,Y 362.075,Z 891.917,A -85,B 0,C 180,E1 -13140,E2 -13140} C_VEL
LIN {X 0,Y 362.052,Z 891.01,A -85,B 0,C 180,E1 -13141.112,E2 -13141.112} C_VEL
LIN {X 0,Y 361.928,Z 889.765,A -85,B 0,C 180,E1 -13142.226,E2 -13142.226} C_VEL
LIN {X 0,Y 361.87,Z 887.021,A -85,B 0,C 180,E1 -13143.898,E2 -13143.898} C_VEL
LIN {X 0,Y 362.212,Z 883.186,A -85,B 0,C 180,E1 -13145.567,E2 -13145.567} C_VEL
LIN {X 0,Y 362.549,Z 877.176,A -85,B 0,C 180,E1 -13147.519,E2 -13147.519} C_VEL
LIN {X 0,Y 362.887,Z 871.584,A -85,B 0,C 180,E1 -13148.97,E2 -13148.97} C_VEL
LIN {X 0,Y 363.235,Z 865.393,A -85,B 0,C 180,E1 -13150.31,E2 -13150.31} C_VEL
LIN {X 0,Y 363.707,Z 857.623,A -85,B 0,C 180,E1 -13151.706,E2 -13151.706} C_VEL
LIN {X 0,Y 364.127,Z 849.252,A -85,B 0,C 180,E1 -13152.966,E2 -13152.966} C_VEL
LIN {X 0,Y 364.626,Z 840.38,A -85,B 0,C 180,E1 -13154.084,E2 -13154.084} C_VEL
LIN {X 0,Y 365.123,Z 831.104,A -85,B 0,C 180,E1 -13155.061,E2 -13155.061} C_VEL
LIN {X 0,Y 365.546,Z 821.56,A -85,B 0,C 180,E1 -13155.897,E2 -13155.897} C_VEL
LIN {X 0,Y 365.896,Z 811.62,A -85,B 0,C 180,E1 -13156.61,E2 -13156.61} C_VEL
LIN {X 0,Y 366.161,Z 801.292,A -85,B 0,C 180,E1 -13157.2,E2 -13157.2} C_VEL
LIN {X 0,Y 366.357,Z 790.694,A -85,B 0,C 180,E1 -13157.658,E2 -13157.658} C_VEL
LIN {X 0,Y 366.531,Z 777.038,A -85,B 0,C 180,E1 -13158.067,E2 -13158.067} C_VEL
LIN {X 0,Y 367.489,Z 724.545,A -85,B 0,C 180,E1 -13159.36,E2 -13159.36} C_VEL
LIN {X 0,Y 361.909,Z 707.403,A -85,B 0,C 180,E1 -13160.069,E2 -13160.069} C_VEL
LIN {X 0,Y 361.915,Z 707.401,A -85,B 0,C 180,E1 -13164.111,E2 -13164.111} C_VEL
LIN {X 0,Y 361.863,Z 707.405,A -85,B 0,C 180,E1 -13167.783,E2 -13167.783} C_VEL
LIN {X 0,Y 361.866,Z 707.409,A -85,B 0,C 180,E1 -13171.283,E2 -13171.283} C_VEL
LIN {X 0,Y 361.871,Z 707.405,A -85,B 0,C 180,E1 -13174.279,E2 -13174.279} C_VEL
LIN {X 0,Y 361.878,Z 707.407,A -85,B 0,C 180,E1 -13177.219,E2 -13177.219} C_VEL
LIN {X 0,Y 361.831,Z 707.413,A -85,B 0,C 180,E1 -13180.748,E2 -13180.748} C_VEL
LIN {X 0,Y 361.831,Z 707.407,A -85,B 0,C 180,E1 -13184.367,E2 -13184.367} C_VEL
LIN {X 0,Y 361.842,Z 707.407,A -85,B 0,C 180,E1 -13187.568,E2 -13187.568} C_VEL
LIN {X 0,Y 361.861,Z 707.405,A -85,B 0,C 180,E1 -13191.568,E2 -13191.568} C_VEL
LIN {X 0,Y 361.888,Z 707.402,A -85,B 0,C 180,E1 -13194.653,E2 -13194.653} C_VEL
LIN {X 0,Y 361.864,Z 707.406,A -85,B 0,C 180,E1 -13197.051,E2 -13197.051} C_VEL
LIN {X 0,Y 361.867,Z 707.406,A -85,B 0,C 180,E1 -13200.946,E2 -13200.946} C_VEL
LIN {X 0,Y 361.866,Z 707.408,A -85,B 0,C 180,E1 -13204.699,E2 -13204.699} C_VEL
LIN {X 0,Y 361.904,Z 707.405,A -85,B 0,C 180,E1 -13208.267,E2 -13208.267} C_VEL
LIN {X 0,Y 363.313,Z 711.297,A -85,B 0,C 180,E1 -13208.457,E2 -13208.457} C_VEL
LIN {X 0,Y 370.686,Z 728.656,A -85,B 0,C 180,E1 -13209.285,E2 -13209.285} C_VEL
LIN {X 0,Y 370.071,Z 786.685,A -85,B 0,C 180,E1 -13210.437,E2 -13210.437} C_VEL
LIN {X 0,Y 370.034,Z 800.314,A -85,B 0,C 180,E1 -13210.882,E2 -13210.882} C_VEL
LIN {X 0,Y 369.662,Z 812.546,A -85,B 0,C 180,E1 -13211.497,E2 -13211.497} C_VEL
LIN {X 0,Y 369.051,Z 823.686,A -85,B 0,C 180,E1 -13212.254,E2 -13212.254} C_VEL
LIN {X 0,Y 368.286,Z 835.054,A -85,B 0,C 180,E1 -13213.256,E2 -13213.256} C_VEL
LIN {X 0,Y 367.46,Z 844.728,A -85,B 0,C 180,E1 -13214.32,E2 -13214.32} C_VEL
LIN {X 0,Y 366.617,Z 853.929,A -85,B 0,C 180,E1 -13215.563,E2 -13215.563} C_VEL
LIN {X 0,Y 365.754,Z 862.307,A -85,B 0,C 180,E1 -13216.945,E2 -13216.945} C_VEL
LIN {X 0,Y 364.738,Z 870.441,A -85,B 0,C 180,E1 -13218.602,E2 -13218.602} C_VEL
LIN {X 0,Y 363.929,Z 877.306,A -85,B 0,C 180,E1 -13220.361,E2 -13220.361} C_VEL
LIN {X 0,Y 363.377,Z 882.929,A -85,B 0,C 180,E1 -13222.212,E2 -13222.212} C_VEL
LIN {X 0,Y 362.739,Z 886.824,A -85,B 0,C 180,E1 -13223.876,E2 -13223.876} C_VEL
LIN {X 0,Y 362.317,Z 889.69,A -85,B 0,C 180,E1 -13225.543,E2 -13225.543} C_VEL
LIN {X 0,Y 362.245,Z 891.05,A -85,B 0,C 180,E1 -13226.656,E2 -13226.656} C_VEL
LIN {X 0,Y 362.235,Z 892.009,A -85,B 0,C 180,E1 -13227.769,E2 -13227.769} C_VEL
LIN {X 0,Y 362.07,Z 892.852,A -85,B 0,C 180,E1 -13229.993,E2 -13229.993} C_VEL
LIN {X 0,Y 362.245,Z 892.091,A -85,B 0,C 180,E1 -13232.216,E2 -13232.216} C_VEL
LIN {X 0,Y 362.302,Z 889.861,A -85,B 0,C 180,E1 -13234.443,E2 -13234.443} C_VEL
LIN {X 0,Y 362.728,Z 887.049,A -85,B 0,C 180,E1 -13236.109,E2 -13236.109} C_VEL
LIN {X 0,Y 363.347,Z 883.225,A -85,B 0,C 180,E1 -13237.774,E2 -13237.774} C_VEL
LIN {X 0,Y 363.903,Z 877.755,A -85,B 0,C 180,E1 -13239.615,E2 -13239.615} C_VEL
LIN {X 0,Y 364.737,Z 870.802,A -85,B 0,C 180,E1 -13241.416,E2 -13241.416} C_VEL
LIN {X 0,Y 365.721,Z 862.921,A -85,B 0,C 180,E1 -13243.041,E2 -13243.041} C_VEL
LIN {X 0,Y 366.578,Z 854.706,A -85,B 0,C 180,E1 -13244.424,E2 -13244.424} C_VEL
LIN {X 0,Y 366.949,Z 850.599,A -85,B 0,C 180,E1 -13245.021,E2 -13245.021} C_VEL
LIN {X 0,Y 366.572,Z 847.714,A -85,B 0,C 180,E1 -13245.451,E2 -13245.451} C_VEL
LIN {X 0,Y 361.995,Z 838.686,A -85,B 0,C 180,E1 -13246.86,E2 -13246.86} C_VEL
LIN {X 0,Y 361.701,Z 835.452,A -85,B 0,C 180,E1 -13247.226,E2 -13247.226} C_VEL
LIN {X 0,Y 362.422,Z 825.036,A -85,B 0,C 180,E1 -13248.158,E2 -13248.158} C_VEL
LIN {X 0,Y 363.093,Z 813.479,A -85,B 0,C 180,E1 -13248.96,E2 -13248.96} C_VEL
LIN {X 0,Y 363.427,Z 801.253,A -85,B 0,C 180,E1 -13249.587,E2 -13249.587} C_VEL
LIN {X 0,Y 363.548,Z 789.667,A -85,B 0,C 180,E1 -13249.985,E2 -13249.985} C_VEL
LIN {X 0,Y 363.861,Z 751.341,A -85,B 0,C 180,E1 -13250.778,E2 -13250.778} C_VEL
LIN {X 0,Y 364.22,Z 730.603,A -85,B 0,C 180,E1 -13251.187,E2 -13251.187} C_VEL
LIN {X 0,Y 354.936,Z 708.828,A -85,B 0,C 180,E1 -13252.268,E2 -13252.268} C_VEL
LIN {X 0,Y 354.845,Z 708.276,A -85,B 0,C 180,E1 -13252.325,E2 -13252.325} C_VEL
LIN {X 0,Y 354.875,Z 708.273,A -85,B 0,C 180,E1 -13255.819,E2 -13255.819} C_VEL
LIN {X 0,Y 354.79,Z 708.287,A -85,B 0,C 180,E1 -13259.673,E2 -13259.673} C_VEL
LIN {X 0,Y 354.774,Z 708.291,A -85,B 0,C 180,E1 -13263.694,E2 -13263.694} C_VEL
LIN {X 0,Y 354.764,Z 708.292,A -85,B 0,C 180,E1 -13266.451,E2 -13266.451} C_VEL
LIN {X 0,Y 354.786,Z 708.28,A -85,B 0,C 180,E1 -13269.416,E2 -13269.416} C_VEL
LIN {X 0,Y 354.8,Z 708.29,A -85,B 0,C 180,E1 -13272.869,E2 -13272.869} C_VEL
LIN {X 0,Y 354.822,Z 708.273,A -85,B 0,C 180,E1 -13276.112,E2 -13276.112} C_VEL
LIN {X 0,Y 354.808,Z 708.29,A -85,B 0,C 180,E1 -13279.181,E2 -13279.181} C_VEL
LIN {X 0,Y 354.757,Z 708.294,A -85,B 0,C 180,E1 -13282.396,E2 -13282.396} C_VEL
LIN {X 0,Y 354.757,Z 708.289,A -85,B 0,C 180,E1 -13284.934,E2 -13284.934} C_VEL
LIN {X 0,Y 354.757,Z 708.294,A -85,B 0,C 180,E1 -13288.394,E2 -13288.394} C_VEL
LIN {X 0,Y 354.791,Z 708.281,A -85,B 0,C 180,E1 -13291.614,E2 -13291.614} C_VEL
LIN {X 0,Y 354.837,Z 708.286,A -85,B 0,C 180,E1 -13294.168,E2 -13294.168} C_VEL
LIN {X 0,Y 354.771,Z 708.287,A -85,B 0,C 180,E1 -13297.89,E2 -13297.89} C_VEL
LIN {X 0,Y 354.856,Z 708.276,A -85,B 0,C 180,E1 -13301.888,E2 -13301.888} C_VEL
LIN {X 0,Y 354.875,Z 708.279,A -85,B 0,C 180,E1 -13305.979,E2 -13305.979} C_VEL
LIN {X 0,Y 354.913,Z 708.264,A -85,B 0,C 180,E1 -13309.734,E2 -13309.734} C_VEL
LIN {X 0,Y 355.06,Z 708.259,A -85,B 0,C 180,E1 -13313.179,E2 -13313.179} C_VEL
LIN {X 0,Y 355.182,Z 708.24,A -85,B 0,C 180,E1 -13317.732,E2 -13317.732} C_VEL
LIN {X 0,Y 355.327,Z 708.224,A -85,B 0,C 180,E1 -13320,E2 -13320} C_VEL
LIN {X 0,Y 355.182,Z 708.235,A -85,B 0,C 180,E1 -13322.268,E2 -13322.268} C_VEL
LIN {X 0,Y 355.06,Z 708.26,A -85,B 0,C 180,E1 -13326.821,E2 -13326.821} C_VEL
LIN {X 0,Y 354.913,Z 708.269,A -85,B 0,C 180,E1 -13330.266,E2 -13330.266} C_VEL
LIN {X 0,Y 354.874,Z 708.278,A -85,B 0,C 180,E1 -13334.021,E2 -13334.021} C_VEL
LIN {X 0,Y 354.856,Z 708.281,A -85,B 0,C 180,E1 -13338.112,E2 -13338.112} C_VEL
LIN {X 0,Y 354.765,Z 708.292,A -85,B 0,C 180,E1 -13342.111,E2 -13342.111} C_VEL
LIN {X 0,Y 354.837,Z 708.277,A -85,B 0,C 180,E1 -13345.832,E2 -13345.832} C_VEL
LIN {X 0,Y 354.796,Z 708.286,A -85,B 0,C 180,E1 -13349.684,E2 -13349.684} C_VEL
LIN {X 0,Y 354.775,Z 708.29,A -85,B 0,C 180,E1 -13353.688,E2 -13353.688} C_VEL
LIN {X 0,Y 354.748,Z 708.294,A -85,B 0,C 180,E1 -13356.466,E2 -13356.466} C_VEL
LIN {X 0,Y 354.774,Z 708.278,A -85,B 0,C 180,E1 -13359.43,E2 -13359.43} C_VEL
LIN {X 0,Y 354.794,Z 708.289,A -85,B 0,C 180,E1 -13362.884,E2 -13362.884} C_VEL
LIN {X 0,Y 354.824,Z 708.289,A -85,B 0,C 180,E1 -13366.127,E2 -13366.127} C_VEL
LIN {X 0,Y 354.816,Z 708.289,A -85,B 0,C 180,E1 -13369.196,E2 -13369.196} C_VEL
LIN {X 0,Y 354.776,Z 708.294,A -85,B 0,C 180,E1 -13372.409,E2 -13372.409} C_VEL
LIN {X 0,Y 354.797,Z 708.397,A -85,B 0,C 180,E1 -13374.041,E2 -13374.041} C_VEL
LIN {X 0,Y 357.777,Z 720.306,A -85,B 0,C 180,E1 -13376.643,E2 -13376.643} C_VEL
LIN {X 0,Y 360.967,Z 734.631,A -85,B 0,C 180,E1 -13379.599,E2 -13379.599} C_VEL
LIN {X 0,Y 361.421,Z 738.149,A -85,B 0,C 180,E1 -13380.284,E2 -13380.284} C_VEL
LIN {X 0,Y 359.41,Z 757.848,A -85,B 0,C 180,E1 -13383.801,E2 -13383.801} C_VEL
LIN {X 0,Y 357.578,Z 778.267,A -85,B 0,C 180,E1 -13387.431,E2 -13387.431} C_VEL
LIN {X 0,Y 361.819,Z 815.903,A -85,B 0,C 180,E1 -13388.479,E2 -13388.479} C_VEL
LIN {X 0,Y 362.992,Z 830.306,A -85,B 0,C 180,E1 -13388.846,E2 -13388.846} C_VEL
LIN {X 0,Y 361.763,Z 889.217,A -85,B 0,C 180,E1 -13390.023,E2 -13390.023} C_VEL
LIN {X 0,Y 361.143,Z 902.41,A -85,B 0,C 180,E1 -13390.506,E2 -13390.506} C_VEL
LIN {X 0,Y 360.152,Z 914.561,A -85,B 0,C 180,E1 -13391.153,E2 -13391.153} C_VEL
LIN {X 0,Y 358.965,Z 926.879,A -85,B 0,C 180,E1 -13392.049,E2 -13392.049} C_VEL
LIN {X 0,Y 357.716,Z 938.565,A -85,B 0,C 180,E1 -13393.164,E2 -13393.164} C_VEL
LIN {X 0,Y 356.706,Z 948.044,A -85,B 0,C 180,E1 -13394.291,E2 -13394.291} C_VEL
LIN {X 0,Y 355.672,Z 957.549,A -85,B 0,C 180,E1 -13395.668,E2 -13395.668} C_VEL
LIN {X 0,Y 355.33,Z 962.82,A -85,B 0,C 180,E1 -13396.57,E2 -13396.57} C_VEL
LIN {X 0,Y 354.596,Z 970.008,A -85,B 0,C 180,E1 -13397.997,E2 -13397.997} C_VEL
LIN {X 0,Y 354.122,Z 977.101,A -85,B 0,C 180,E1 -13399.719,E2 -13399.719} C_VEL
LIN {X 0,Y 353.916,Z 982.818,A -85,B 0,C 180,E1 -13401.443,E2 -13401.443} C_VEL
LIN {X 0,Y 353.982,Z 988.034,A -85,B 0,C 180,E1 -13403.471,E2 -13403.471} C_VEL
LIN {X 0,Y 354.108,Z 991.691,A -85,B 0,C 180,E1 -13405.454,E2 -13405.454} C_VEL
LIN {X 0,Y 354.186,Z 993.156,A -85,B 0,C 180,E1 -13406.595,E2 -13406.595} C_VEL
LIN {X 0,Y 354.231,Z 994.197,A -85,B 0,C 180,E1 -13407.734,E2 -13407.734} C_VEL
LIN {X 0,Y 354.298,Z 994.837,A -85,B 0,C 180,E1 -13408.871,E2 -13408.871} C_VEL
LIN {X 0,Y 354.357,Z 995.065,A -85,B 0,C 180,E1 -13410.008,E2 -13410.008} C_VEL
LIN {X 0,Y 354.299,Z 994.826,A -85,B 0,C 180,E1 -13411.144,E2 -13411.144} C_VEL
LIN {X 0,Y 354.232,Z 994.179,A -85,B 0,C 180,E1 -13412.281,E2 -13412.281} C_VEL
LIN {X 0,Y 354.189,Z 993.129,A -85,B 0,C 180,E1 -13413.42,E2 -13413.42} C_VEL
LIN {X 0,Y 354.11,Z 991.654,A -85,B 0,C 180,E1 -13414.561,E2 -13414.561} C_VEL
LIN {X 0,Y 353.945,Z 988.129,A -85,B 0,C 180,E1 -13416.477,E2 -13416.477} C_VEL
LIN {X 0,Y 353.925,Z 982.75,A -85,B 0,C 180,E1 -13418.572,E2 -13418.572} C_VEL
LIN {X 0,Y 354.129,Z 977.013,A -85,B 0,C 180,E1 -13420.296,E2 -13420.296} C_VEL
LIN {X 0,Y 354.611,Z 969.901,A -85,B 0,C 180,E1 -13422.018,E2 -13422.018} C_VEL
LIN {X 0,Y 355.324,Z 962.687,A -85,B 0,C 180,E1 -13423.445,E2 -13423.445} C_VEL
LIN {X 0,Y 355.649,Z 957.222,A -85,B 0,C 180,E1 -13424.374,E2 -13424.374} C_VEL
LIN {X 0,Y 356.724,Z 947.855,A -85,B 0,C 180,E1 -13425.724,E2 -13425.724} C_VEL
LIN {X 0,Y 357.722,Z 938.331,A -85,B 0,C 180,E1 -13426.852,E2 -13426.852} C_VEL
LIN {X 0,Y 358.966,Z 926.588,A -85,B 0,C 180,E1 -13427.967,E2 -13427.967} C_VEL
LIN {X 0,Y 360.177,Z 914.159,A -85,B 0,C 180,E1 -13428.862,E2 -13428.862} C_VEL
LIN {X 0,Y 361.658,Z 895.824,A -85,B 0,C 180,E1 -13429.814,E2 -13429.814} C_VEL
LIN {X 0,Y 362.435,Z 883.942,A -85,B 0,C 180,E1 -13430.287,E2 -13430.287} C_VEL
LIN {X 0,Y 364.842,Z 826.961,A -85,B 0,C 180,E1 -13431.944,E2 -13431.944} C_VEL
LIN {X 0,Y 363.063,Z 798.447,A -85,B 0,C 180,E1 -13433.115,E2 -13433.115} C_VEL
LIN {X 0,Y 360.621,Z 778.712,A -85,B 0,C 180,E1 -13434.104,E2 -13434.104} C_VEL
LIN {X 0,Y 358.676,Z 765.364,A -85,B 0,C 180,E1 -13434.844,E2 -13434.844} C_VEL
LIN {X 0,Y 360.807,Z 744.057,A -85,B 0,C 180,E1 -13438.646,E2 -13438.646} C_VEL
LIN {X 0,Y 361.359,Z 737.959,A -85,B 0,C 180,E1 -13439.738,E2 -13439.738} C_VEL
LIN {X 0,Y 359.701,Z 728.771,A -85,B 0,C 180,E1 -13441.573,E2 -13441.573} C_VEL
LIN {X 0,Y 356.227,Z 713.956,A -85,B 0,C 180,E1 -13444.707,E2 -13444.707} C_VEL
LIN {X 0,Y 354.807,Z 708.273,A -85,B 0,C 180,E1 -13445.977,E2 -13445.977} C_VEL
LIN {X 0,Y 354.788,Z 708.293,A -85,B 0,C 180,E1 -13449.416,E2 -13449.416} C_VEL
LIN {X 0,Y 354.785,Z 708.289,A -85,B 0,C 180,E1 -13452.866,E2 -13452.866} C_VEL
LIN {X 0,Y 354.774,Z 708.291,A -85,B 0,C 180,E1 -13456.105,E2 -13456.105} C_VEL
LIN {X 0,Y 354.782,Z 708.291,A -85,B 0,C 180,E1 -13459.178,E2 -13459.178} C_VEL
LIN {X 0,Y 354.818,Z 708.285,A -85,B 0,C 180,E1 -13462.407,E2 -13462.407} C_VEL
LIN {X 0,Y 354.828,Z 708.284,A -85,B 0,C 180,E1 -13464.942,E2 -13464.942} C_VEL
LIN {X 0,Y 354.81,Z 708.286,A -85,B 0,C 180,E1 -13468.409,E2 -13468.409} C_VEL
LIN {X 0,Y 354.82,Z 708.287,A -85,B 0,C 180,E1 -13471.616,E2 -13471.616} C_VEL
LIN {X 0,Y 354.864,Z 708.282,A -85,B 0,C 180,E1 -13474.801,E2 -13474.801} C_VEL
LIN {X 0,Y 355.853,Z 711.112,A -85,B 0,C 180,E1 -13475.085,E2 -13475.085} C_VEL
LIN {X 0,Y 357.524,Z 713.326,A -85,B 0,C 180,E1 -13475.426,E2 -13475.426} C_VEL
LIN {X 0,Y 359.518,Z 716.641,A -85,B 0,C 180,E1 -13475.855,E2 -13475.855} C_VEL
LIN {X 0,Y 366.274,Z 729.171,A -85,B 0,C 180,E1 -13477.217,E2 -13477.217} C_VEL
LIN {X 0,Y 368.534,Z 733.898,A -85,B 0,C 180,E1 -13477.648,E2 -13477.648} C_VEL
LIN {X 0,Y 365.907,Z 788.258,A -85,B 0,C 180,E1 -13479.297,E2 -13479.297} C_VEL
LIN {X 0,Y 365.691,Z 801.968,A -85,B 0,C 180,E1 -13479.798,E2 -13479.798} C_VEL
LIN {X 0,Y 365.326,Z 812.526,A -85,B 0,C 180,E1 -13480.327,E2 -13480.327} C_VEL
LIN {X 0,Y 364.757,Z 823.464,A -85,B 0,C 180,E1 -13481.044,E2 -13481.044} C_VEL
LIN {X 0,Y 363.942,Z 834.953,A -85,B 0,C 180,E1 -13482.003,E2 -13482.003} C_VEL
LIN {X 0,Y 362.795,Z 846.508,A -85,B 0,C 180,E1 -13483.252,E2 -13483.252} C_VEL
LIN {X 0,Y 362.052,Z 853.992,A -85,B 0,C 180,E1 -13484.231,E2 -13484.231} C_VEL
LIN {X 0,Y 361.166,Z 861.26,A -85,B 0,C 180,E1 -13485.347,E2 -13485.347} C_VEL
LIN {X 0,Y 360.155,Z 868.767,A -85,B 0,C 180,E1 -13486.745,E2 -13486.745} C_VEL
LIN {X 0,Y 359.23,Z 874.97,A -85,B 0,C 180,E1 -13488.146,E2 -13488.146} C_VEL
LIN {X 0,Y 358.513,Z 879.219,A -85,B 0,C 180,E1 -13489.267,E2 -13489.267} C_VEL
LIN {X 0,Y 357.619,Z 884.312,A -85,B 0,C 180,E1 -13490.955,E2 -13490.955} C_VEL
LIN {X 0,Y 356.824,Z 888.194,A -85,B 0,C 180,E1 -13492.645,E2 -13492.645} C_VEL
LIN {X 0,Y 356.218,Z 890.955,A -85,B 0,C 180,E1 -13494.339,E2 -13494.339} C_VEL
LIN {X 0,Y 355.965,Z 892.274,A -85,B 0,C 180,E1 -13495.47,E2 -13495.47} C_VEL
LIN {X 0,Y 355.434,Z 893.47,A -85,B 0,C 180,E1 -13497.734,E2 -13497.734} C_VEL
LIN {X 0,Y 355.249,Z 893.443,A -85,B 0,C 180,E1 -13498.866,E2 -13498.866} C_VEL
LIN {X 0,Y 355.054,Z 892.963,A -85,B 0,C 180,E1 -13500,E2 -13500} C_VEL
LIN {X 0,Y 354.902,Z 890.704,A -85,B 0,C 180,E1 -13502.27,E2 -13502.27} C_VEL
LIN {X 0,Y 354.846,Z 887.839,A -85,B 0,C 180,E1 -13503.975,E2 -13503.975} C_VEL
LIN {X 0,Y 355.202,Z 883.859,A -85,B 0,C 180,E1 -13505.678,E2 -13505.678} C_VEL
LIN {X 0,Y 355.536,Z 877.664,A -85,B 0,C 180,E1 -13507.668,E2 -13507.668} C_VEL
LIN {X 0,Y 355.852,Z 872.175,A -85,B 0,C 180,E1 -13509.091,E2 -13509.091} C_VEL
LIN {X 0,Y 356.23,Z 865.575,A -85,B 0,C 180,E1 -13510.515,E2 -13510.515} C_VEL
LIN {X 0,Y 356.616,Z 859.394,A -85,B 0,C 180,E1 -13511.654,E2 -13511.654} C_VEL
LIN {X 0,Y 357.114,Z 850.107,A -85,B 0,C 180,E1 -13513.081,E2 -13513.081} C_VEL
LIN {X 0,Y 357.517,Z 842.435,A -85,B 0,C 180,E1 -13514.079,E2 -13514.079} C_VEL
LIN {X 0,Y 358.073,Z 833.376,A -85,B 0,C 180,E1 -13515.074,E2 -13515.074} C_VEL
LIN {X 0,Y 358.567,Z 823.041,A -85,B 0,C 180,E1 -13516.011,E2 -13516.011} C_VEL
LIN {X 0,Y 358.937,Z 812.784,A -85,B 0,C 180,E1 -13516.768,E2 -13516.768} C_VEL
LIN {X 0,Y 359.184,Z 802.014,A -85,B 0,C 180,E1 -13517.398,E2 -13517.398} C_VEL
LIN {X 0,Y 359.411,Z 791.419,A -85,B 0,C 180,E1 -13517.864,E2 -13517.864} C_VEL
LIN {X 0,Y 359.588,Z 777.695,A -85,B 0,C 180,E1 -13518.282,E2 -13518.282} C_VEL
LIN {X 0,Y 360.56,Z 725.963,A -85,B 0,C 180,E1 -13519.595,E2 -13519.595} C_VEL
LIN {X 0,Y 354.853,Z 708.284,A -85,B 0,C 180,E1 -13520.338,E2 -13520.338} C_VEL
LIN {X 0,Y 354.856,Z 708.282,A -85,B 0,C 180,E1 -13524.341,E2 -13524.341} C_VEL
LIN {X 0,Y 354.821,Z 708.284,A -85,B 0,C 180,E1 -13528.384,E2 -13528.384} C_VEL
LIN {X 0,Y 354.805,Z 708.287,A -85,B 0,C 180,E1 -13532.332,E2 -13532.332} C_VEL
LIN {X 0,Y 354.839,Z 708.28,A -85,B 0,C 180,E1 -13535.696,E2 -13535.696} C_VEL
LIN {X 0,Y 354.79,Z 708.288,A -85,B 0,C 180,E1 -13539.41,E2 -13539.41} C_VEL
LIN {X 0,Y 354.801,Z 708.288,A -85,B 0,C 180,E1 -13542.863,E2 -13542.863} C_VEL
LIN {X 0,Y 354.782,Z 708.285,A -85,B 0,C 180,E1 -13546.099,E2 -13546.099} C_VEL
LIN {X 0,Y 354.782,Z 708.288,A -85,B 0,C 180,E1 -13549.172,E2 -13549.172} C_VEL
LIN {X 0,Y 354.817,Z 708.281,A -85,B 0,C 180,E1 -13552.401,E2 -13552.401} C_VEL
LIN {X 0,Y 354.826,Z 708.282,A -85,B 0,C 180,E1 -13554.936,E2 -13554.936} C_VEL
LIN {X 0,Y 354.794,Z 708.285,A -85,B 0,C 180,E1 -13558.406,E2 -13558.406} C_VEL
LIN {X 0,Y 354.805,Z 708.286,A -85,B 0,C 180,E1 -13561.609,E2 -13561.609} C_VEL
LIN {X 0,Y 354.817,Z 708.287,A -85,B 0,C 180,E1 -13565.414,E2 -13565.414} C_VEL
LIN {X 0,Y 354.864,Z 708.464,A -85,B 0,C 180,E1 -13567.827,E2 -13567.827} C_VEL
LIN {X 0,Y 356.701,Z 713.138,A -85,B 0,C 180,E1 -13568.054,E2 -13568.054} C_VEL
LIN {X 0,Y 364.144,Z 730.599,A -85,B 0,C 180,E1 -13568.914,E2 -13568.914} C_VEL
LIN {X 0,Y 363.447,Z 786.775,A -85,B 0,C 180,E1 -13570.043,E2 -13570.043} C_VEL
LIN {X 0,Y 363.393,Z 800.59,A -85,B 0,C 180,E1 -13570.489,E2 -13570.489} C_VEL
